// TIA Portal V20 export
// export: Created 2025-12-01T14:57:12.8919751Z, ExportSetting None, DisplayName Totally Integrated Automation Portal, DisplayVersion V20 Update 3, DisplayName TIA Portal Openness, DisplayVersion V20 Update 3, DisplayName TIA Portal Version Control Interface, DisplayVersion V20 Update 3, DisplayName STEP 7 Professional, DisplayVersion V20 Update 3, DisplayName STEP 7 Safety, DisplayVersion V20 Update 2, DisplayName WinCC Basic/Comfort/Advanced, DisplayVersion V20 Update 3, DisplayName WinCC Professional, DisplayVersion V20 Update 3, DisplayName WinCC Unified, DisplayVersion V20 Update 3
FUNCTION "FC811_EventosGenerados" : Void   // FC811, LAD
TITLE = "EventosGenerados" - Se generar la lista de Eventos a Emitir
{ S7_Optimized_Access := 'FALSE' }
AUTHOR : TRACKING
NAME : 20160407
VERSION : 4.2
// - Inicializaciones
// - Mirar si se pueden generar eventos
// - Generar eventos de las UT's
// - Generar eventos de los dispositivos
// - Generar eventos de las Mesas
// stored: AutoNumber false, SetENOAutomatically false
   VAR_INPUT
      NumJdT : UInt;
   END_VAR
   VAR_TEMP
      DBEventos : Word;   // Num. DB de eventos generados
      NumDBEventos : UInt;
      P_Eventos : DWord;   // Puntero al DB de Eventos Generados
      MaxBytes : UInt;
      InicioBucleMesas : UInt;
      FinalBucleMesas : UInt;
      NumBytes : UInt;   // Numero de Bytes a Emitir
      P_Temporal : DWord;
      NumMesa : UInt;   // Numero de Mesa a mirar
      IndiceEtiqueta : UInt;
      NumeroUT : UInt;   // Numero de UT a mirar
      EventoUT : UInt;   // Numero de Evento Generado en la UT
      EventoDispositivo : UInt;   // Numero de Evento Genarado en el Dispositivo
      NivelPantalla : UInt;   // Numero de nivel de pantalla
      Convertir : UInt;
      Conversion : DWord;
      Valor : UDInt;
      Offset : UInt;
      Proceso : UInt;
      ResultadoProceso : UInt;
      ValorReturn : Int;
      MesaDeJDT02 : Bool;
      JDT02_Activo : Bool;
      DispoDeJDT02 : Bool;
   END_VAR
BEGIN

NETWORK
TITLE = Inicializaciones
// - Inicializar las variables de los DB's
////////////////////////////////////////////////////////////////////////////////
////////////////////////////////////////////////////////////////////////////////
/// Inicio Que conexion es de JDT

      SET;
      R     #JDT02_Activo;
      L     "JDT1_NDB_EventosEmi";
      T     #DBEventos;
      T     #NumDBEventos;
      L     "JDT2_MaxBytes";
      T     #MaxBytes;

      L     "JDT1_InicioBucleMesas";  // Tamaño Bucles
      T     #InicioBucleMesas;
      L     "JDT1_FinalBucleMesas";
      T     #FinalBucleMesas;

      L     #NumJdT;
      L     2;
      <>I;
      JC    NoJDT02;

      SET;
      S     #JDT02_Activo;
      L     "JDT2_NDB_EventosEmi";
      T     #DBEventos;
      T     #NumDBEventos;
      L     "JDT2_MaxBytes";
      T     #MaxBytes;

      L     "JDT2_InicioBucleMesas";  // Tamaño Bucles
      T     #InicioBucleMesas;
      L     "JDT2_FinalBucleMesas";
      T     #FinalBucleMesas;

NoJDT02:NOP   0;

/// FIn Que conexion es de JDT
////////////////////////////////////////////////////////////////////////////////
////////////////////////////////////////////////////////////////////////////////



NETWORK
TITLE = Mirar si se pueden generar eventos
// - Inicializo el Numero de Bytes y el puntero del DB de Eventos Generados
// - Calcula el Tamaño de bytes que hay en el DB de Eventos Genardos
// - Comprobamos si hay sitio para Eventos
////////////////////////////////////////////////////////////////////////////////
// Inicializo el Numero de Bytes y el puntero del DB Eventos Generados

      L     0;
      T     #NumBytes;  // Inicializo el numero de Bytes
      LAR2;  // Inicializo el puntero de Eventos Generados

////////////////////////////////////////////////////////////////////////////////
// Calcula el tamaño de bytes que hay en el DB Eventos Generados

      OPN   DB [#DBEventos];

InicioBucleBusquedaFin_BufferEventos:NOP   0;
      L     DBB [AR2, P#0.0];
      L     0;
      ==I;
      JC    FinBucleBusquedaFin_BufferEventos;  // Buscamos el final del DB = 0

      +AR2  P#1.0;
      JU    InicioBucleBusquedaFin_BufferEventos;

FinBucleBusquedaFin_BufferEventos:NOP   0;
      TAR2;  // Guardo el puntero
      T     #P_Eventos;  // Sacamos el NumBytes Escritos
      SRD   3;
      T     #NumBytes;

////////////////////////////////////////////////////////////////////////////////
// Comprobamos si hay sitio para mas Eventos

      L     #NumBytes;  // Miramos si hay sitio
      L     #MaxBytes;  // Max. que se pueden emitir, parametro
      >I;
      JC    FinalFuncion;  // No se pueden generar más eventos



NETWORK
TITLE = Generar Eventos de las UT's
// - Recorrer todas las Mesas Buscando UT'que necesiten generar Eventos
//   Dos bucles anidados Mesas y UT's dentro de las Mesas ( No se hace)
// - Recorrer todas las UT's (Se hace
////////////////////////////////////////////////////////////////////////////////
////////////////////////////////////////////////////////////////////////////////
////////////////////////////////////////////////////////////////////////////////
// Recorrer todas las Mesas

      L     #InicioBucleMesas;
      T     #NumMesa;

InicioBucleMesa_EventosUT:NOP   0;
////////////////////////////////////////////////////////////////////////////////
/// Mirar Si pertenece al JDT

      SET;
      X     "DB850_DefinicionMesas".Mesa[#NumMesa].ConfigMesa.MesaDeJDT02;
      XN    #JDT02_Activo;  // JDT01 o JDT02 ?
      =     #MesaDeJDT02;

      SET;
      AN    #MesaDeJDT02;
      JC    ContinuarBucleMesa_EventosUT;

////////////////////////////////////////////////////////////////////////////////
// Mirar si esta definido como mesa de tracking

      SET;
      AN    "DB850_DefinicionMesas".Mesa[#NumMesa].ConfigMesa.MesaPaso;
      AN    "DB850_DefinicionMesas".Mesa[#NumMesa].ConfigMesa.MesaCruce;
      AN    "DB850_DefinicionMesas".Mesa[#NumMesa].ConfigMesa.MesaMultiplesDestinos;
      JC    ContinuarBucleMesa_EventosUT;


////////////////////////////////////////////////////////////////////////////////

      L     "DB810_ColasMesas".Colas[#NumMesa].UT_PrimeraMesa;
      T     #NumeroUT;

      L     #NumeroUT;
      L     0;
      ==I;
      JC    ContinuarBucleMesa_EventosUT;  // No hay UT's en la Mesa


////////////////////////////////////////////////////////////////////////////////
// --- Recorrer todas las UT's de la Mesa
InicioBucleUT_EventosUT:NOP   0;

      L     "DB812_UTs_Control".UT[#NumeroUT].EstadoEventoAGenerar;
      T     #EventoUT;  // Para ver si hay Evento de UT

      L     #EventoUT;  // Mirar si hay evento a generar
      L     100;
      >=I;
      JC    Generar_EventosUT;  // Si es >= 100 Hay evento a generar


////////////////////////////////////////////////////////////////////////////////
ContinuarBucleUT_EventosUT:NOP   0;
      L     "DB812_UTs_Control".UT[#NumeroUT].UT_SiguienteMesa;
      T     #NumeroUT;

      L     #NumeroUT;
      L     0;
      ==I;
      JC    ContinuarBucleMesa_EventosUT;  // No hay mas UT's en la Mesa

      JU    InicioBucleUT_EventosUT;  // Seguir recorriendo la Mesa


////////////////////////////////////////////////////////////////////////////////
// --- Continuar recorriendo el resto de Mesas
ContinuarBucleMesa_EventosUT:NOP   0;
      L     #NumMesa;
      L     #FinalBucleMesas;
      >=I;
      JC    EventosMesa;  // Ya no hay más UT's, recorrer dispositivos

      L     #NumMesa;  // +1, Para la Siguiente UT
      L     1;
      +I;
      T     #NumMesa;

      JU    InicioBucleMesa_EventosUT;  // Ir a mirar la siguiente UT


////////////////////////////////////////////////////////////////////////////////
// Comprobacion del tamaño del DB de Eventos Generados
FinBucles_EventosUT:NOP   0;
      TAR2;
      T     #P_Eventos;
      SRD   3;
      T     #NumBytes;

      L     #NumBytes;  // Miramos si hay sitio
      L     #MaxBytes;
      >I;
      JC    FinalFuncion;  // No se pueden generar más eventos
      JU    ContinuarBucleUT_EventosUT;  // Seguir con las UT's



NETWORK
TITLE = Formatear Eventos de las UTs - Distribucion
Generar_EventosUT:NOP   0;

////////////////////////////////////////////////////////////////////////////////
////////////////////////////////////////////////////////////////////////////////
// -- Formateo del Evento LOCA - Diferentes Motivos (Normal, Reset, Galibo ...)
// -- Formateo del Evento RUT? - Diferentes (Reset, PLC, ...)
// -- Formateo del Evento RET! - Ausencia de la Mesa
// -- Formateo del Evento BOR! - Borrada UT del Sistema
// -- Formateo del Evento DATO - Refresco de Datos de la UT
// -- Formateo del Evento NUUT - Nueva UT en la Mesa
// -- Formateo del Evento DAT? - Peticion de Datos para la UT
// -- Formateo del Evento PEMB (Peticion de Datos de Embandejado de la UT)
////////////////////////////////////////////////////////////////////////////////
////////////////////////////////////////////////////////////////////////////////
// Distribucion para Eventos de las UT's

      L     #EventoUT;  // Formateo del evento
      L     100;  // Presencia Normal
      ==I;
      JC    GenerarEvento_LOCA_EventosUT;

      L     #EventoUT;  // Formateo del evento
      L     101;  // Presencia de Reset
      ==I;
      JC    GenerarEvento_LOCA_EventosUT;

      L     #EventoUT;  // Formateo del evento
      L     102;  // Presencia de Galibo
      ==I;
      JC    GenerarEvento_LOCA_EventosUT;

      L     #EventoUT;  // Formateo del evento
      L     103;  // Ausencia
      ==I;
      JC    GenerarEvento_RET_EventosUT;

      L     #EventoUT;  // Formateo del evento
      L     110;  // Refresco de datos de la UT
      ==I;
      JC    GenerarEvento_DATO_EventoUT;

      L     #EventoUT;  // Formateo del evento
      L     121;  // Peticion de Ruta por MOTIVO --> Reset
      ==I;
      JC    GenerarEvento_RUT_EventoUT;

      L     #EventoUT;  // Formateo del evento
      L     122;  // Peticion de Ruta por MOTIVO --> Bloqueo
      ==I;
      JC    GenerarEvento_RUT_EventoUT;

      L     #EventoUT;  // Formateo del evento
      L     123;  // Peticion de Ruta por MOTIVO --> Llegada a su Destino
      ==I;
      JC    GenerarEvento_RUT_EventoUT;

      L     #EventoUT;  // Formateo del evento
      L     124;  // Peticion de Ruta por MOTIVO --> No tiene Destino
      ==I;
      JC    GenerarEvento_RUT_EventoUT;

      L     #EventoUT;  // Formateo del evento
      L     125;  // Peticion de Ruta por MOTIVO --> Fuera de Ruta
      ==I;
      JC    GenerarEvento_RUT_EventoUT;

      L     #EventoUT;  // Formateo del evento
      L     126;  // Peticion de Ruta por MOTIVO --> Robo de Garra a Elevador
      ==I;
      JC    GenerarEvento_RUT_EventoUT;

      L     #EventoUT;  // Formateo del evento
      L     131;  // Borrar la UT de la Base de datos
      ==I;
      JC    GenerarEvento_BOR_EventosUT;

      L     #EventoUT;  // Formateo del evento
      L     132;  // Nueva UT en la BD
      ==I;
      JC    GenerarEvento_NUUT_EventosUT;

      L     #EventoUT;  // Formateo del evento
      L     141;  // Peticion de datos para la UT
      ==I;
      JC    GenerarEvento_DAT_EventosUT;

      L     #EventoUT;  // Formateo del evento
      L     145;  // Chequeo de la UT >>> Por Reset
      ==I;
      JC    GenerarEvento_CHE_EventosUT;

      L     #EventoUT;  // Formateo del evento     // Fecha 2019 01 18
      L     161;  // Peticion de datos de Embandejado para la UT
      ==I;
      JC    GenerarEvento_PEMB_EventosUT;


////////////////////////////////////////////////////////////////////////////////
////////////////////////////////////////////////////////////////////////////////
////////////////////////////////////////////////////////////////////////////////
// --- Dar por formateado el Evento

      L     0;  // 0 - Dar por Tratado
      T     "DB812_UTs_Control".UT[#NumeroUT].EstadoEventoAGenerar;

      JU    FinBucles_EventosUT;

// Fin de la distribucion para generar los eventos
////////////////////////////////////////////////////////////////////////////////
////////////////////////////////////////////////////////////////////////////////
////////////////////////////////////////////////////////////////////////////////



NETWORK
TITLE = ---- Eventos de UT - Esta en Mesa - LOCA
// - Distribucion para Eventos de las UT's
// - Formateo de Eventos
//   - Evento LOCA (Cambio de Mesa de la UT
//   - Evento RUT? (Petición de Ruta para la UT)
//   - Evento NUUT (Nueva UT en la instalacion)
//   - Evento DATO (Cambio de de datos de la UT)
//   - Evento BOR! (UT Borrada de la Base de datos)
//   - Evento DAT? (Peticion de datos de la UT)
//   - Evento RET! (Retirada de la UT)
GenerarEvento_LOCA_EventosUT:NOP   0;

////////////////////////////////////////////////////////////////////////////////
////////////////////////////////////////////////////////////////////////////////
////////////////////////////////////////////////////////////////////////////////
// -- Formateo del Evento LOCA - Diferentes Motivos (Normal, Reset, Galibo ...)

      L     #P_Eventos;
      LAR2;  // Puntero al DB de Eventos Generados

      TAR2;  // Mirar si es el primer evento de la lista
      L     0;
      ==I;
      JC    InicioBuffer_LOCA_EventosUT;  // Es el primero

      OPN   DB [#DBEventos];  // Hay que añadir si no es el primer evento
      L     ',';  // Separador entre eventos ','
      T     DBB [AR2, P#0.0];
      +AR2  P#1.0;

InicioBuffer_LOCA_EventosUT:NOP   0;
      OPN   DB [#DBEventos];  // DB de Eventos Generados (A Emitir)
      L     '{';  // Inicio de Evento '{'
      T     DBB [AR2, P#0.0];
      +AR2  P#1.0;


////////////////////////////////////////////////////////////////////////////////
      L     'LOCA';  // Evento 'LOCA'
      T     DBD [AR2, P#0.0];
      +AR2  P#4.0;

      L     '[';  // Evento - Atributo Mckey '[MCKY]'
      T     DBB [AR2, P#0.0];
      L     'MCKY';
      T     DBD [AR2, P#1.0];
      L     ']';  // Evento - Atributo Mckey '[MCKY]'
      T     DBB [AR2, P#5.0];
      +AR2  P#6.0;

      L     "DB812_UTs_Control".UT[#NumeroUT].Mckey;
      T     #Valor;

// --- Convertir Valor a ASCII - Mckey
      TAR2;
      SRD   3;
      T     #NumBytes;  // Miro que offset tiene la String

      CALL  "FC893_Obtener_StringDelAtributo"
      ( DB_String := #NumDBEventos,
        OffsetIni := #NumBytes,
        Valor     := #Valor,
        OffsetFin := #Offset
      );  // Llamo a ObtenerStrinAtributo

      L     #Offset;
      SLD   3;
      LAR2;  // Recupero que offset tiene la String

// --- Ya esta convertido el Valor a ASCI - Fin Mckey


////////////////////////////////////////////////////////////////////////////////
      OPN   DB [#DBEventos];
      L     '[';  // Evento - Atributo Mesa Actual '[MESA]'
      T     DBB [AR2, P#0.0];
      L     'MESA';
      T     DBD [AR2, P#1.0];
      L     ']';
      T     DBB [AR2, P#5.0];
      +AR2  P#6.0;

      L     "DB812_UTs_Control".UT[#NumeroUT].MesaActual;
      T     #Valor;

// --- Convertir Valor a ASCII -  Mesa Actual
      TAR2;
      SRD   3;
      T     #NumBytes;  // Miro que offset tiene la String

      CALL  "FC893_Obtener_StringDelAtributo"
      ( DB_String := #NumDBEventos,
        OffsetIni := #NumBytes,
        Valor     := #Valor,
        OffsetFin := #Offset
      );  // Llamo a ObtenerStrinAtributo

      L     #Offset;
      SLD   3;
      LAR2;  // Recupero que offset tiene la String

// --- Ya esta convertido el Valor a ASCI - Fin Mesa Actual


////////////////////////////////////////////////////////////////////////////////
// --- Final del Formateo del Evento ---

      OPN   DB [#DBEventos];  // DB de Eventos Generados (A Emitir)
      L     '}';  // Fin de Evento '}'
      T     DBB [AR2, P#0.0];
      +AR2  P#1.0;



////////////////////////////////////////////////////////////////////////////////
////////////////////////////////////////////////////////////////////////////////
////////////////////////////////////////////////////////////////////////////////
// --- Dar por formateado el Evento

      L     0;  // 0 - Dar por Tratado
      T     "DB812_UTs_Control".UT[#NumeroUT].EstadoEventoAGenerar;

////////////////////////////////////////////////////////////////////////////////
/// Hay que Pedir Datos
      SET;
      AN    "DB812_UTs_Control".UT[#NumeroUT].AtributosDeLaUT.PeticionDeDatos;
      JC    NoPedirDatos_LOCA_EventosUT;

      L     141;
      T     "DB812_UTs_Control".UT[#NumeroUT].EstadoEventoAGenerar;

NoPedirDatos_LOCA_EventosUT:NOP   0;

////////////////////////////////////////////////////////////////////////////////
/// Hay que Generar mas Eventos
      L     #EventoUT;  // Formateo del evento
      L     100;  // Presencia Normal
      ==I;
      JC    FinBucles_EventosUT;

////////////////////////////////////////////////////////////////////////////////
/// Es de Reset de Pantalla, Auto Generar Nuevo Evento
      L     121;  // 121 - Generar evento de Pedir Ruta (Por Reset)
      T     "DB812_UTs_Control".UT[#NumeroUT].EstadoEventoAGenerar;

      L     #EventoUT;  // Formateo del evento
      L     101;  // Presencia de Reset
      ==I;
      JC    FinBucles_EventosUT;


////////////////////////////////////////////////////////////////////////////////
/// Es de Galibo, Auto Generar Nuevo Evento
      L     110;  // Enviar datos de UT
      T     "DB812_UTs_Control".UT[#NumeroUT].EstadoEventoAGenerar;

      JU    FinBucles_EventosUT;

// Fin del Evento LOCA
////////////////////////////////////////////////////////////////////////////////
////////////////////////////////////////////////////////////////////////////////
////////////////////////////////////////////////////////////////////////////////



NETWORK
TITLE = ---- Evento de UT - Peticion de Ruta - RUT?
GenerarEvento_RUT_EventoUT:NOP   0;

////////////////////////////////////////////////////////////////////////////////
////////////////////////////////////////////////////////////////////////////////
////////////////////////////////////////////////////////////////////////////////
////////////////////////////////////////////////////////////////////////////////
// -- Formateo del Evento RUT? - Diferentes (Reset, PLC, ...)

      L     #P_Eventos;
      LAR2;  // Puntero al DB de Eventos Generados

      TAR2;  // Mirar si es el primer evento de la lista
      L     0;
      ==I;
      JC    InicioBuffer_RUT_EventosUT;  // Es el primero

      OPN   DB [#DBEventos];  // Hay que añadir si no es el primer evento
      L     ',';  // Separador entre eventos ','
      T     DBB [AR2, P#0.0];
      +AR2  P#1.0;

InicioBuffer_RUT_EventosUT:NOP   0;
      OPN   DB [#DBEventos];  // DB de Eventos Generados (A Emitir)
      L     '{';  // Inicio de Evento '{'
      T     DBB [AR2, P#0.0];
      +AR2  P#1.0;

      L     'RUT?';  // Evento 'RUT?'
      T     DBD [AR2, P#0.0];
      +AR2  P#4.0;


////////////////////////////////////////////////////////////////////////////////
      L     '[';  // Evento - Atributo Mckey '[MCKEY]'
      T     DBB [AR2, P#0.0];
      L     'MCKY';
      T     DBD [AR2, P#1.0];
      L     ']';
      T     DBB [AR2, P#5.0];
      +AR2  P#6.0;

      L     "DB812_UTs_Control".UT[#NumeroUT].Mckey;
      T     #Valor;

// --- Convertir Valor a ASCII - Mckey
      TAR2;
      SRD   3;
      T     #NumBytes;  // Miro que offset tiene la String

      CALL  "FC893_Obtener_StringDelAtributo"
      ( DB_String := #NumDBEventos,
        OffsetIni := #NumBytes,
        Valor     := #Valor,
        OffsetFin := #Offset
      );  // Llamo a ObtenerStrinAtributo

      L     #Offset;
      SLD   3;
      LAR2;  // Recupero que offset tiene la String

// --- Ya esta convertido el Valor a ASCI - Fin Mckey


////////////////////////////////////////////////////////////////////////////////
      OPN   DB [#DBEventos];
      L     '[';  // Evento - Atributo Mesa Actual '[MESA]'
      T     DBB [AR2, P#0.0];
      L     'MESA';
      T     DBD [AR2, P#1.0];
      L     ']';
      T     DBB [AR2, P#5.0];
      +AR2  P#6.0;

      L     "DB812_UTs_Control".UT[#NumeroUT].MesaActual;
      T     #Valor;

// --- Convertir Valor a ASCII -  Mesa Actual
      TAR2;
      SRD   3;
      T     #NumBytes;  // Miro que offset tiene la String

      CALL  "FC893_Obtener_StringDelAtributo"
      ( DB_String := #NumDBEventos,
        OffsetIni := #NumBytes,
        Valor     := #Valor,
        OffsetFin := #Offset
      );  // Llamo a ObtenerStrinAtributo

      L     #Offset;
      SLD   3;
      LAR2;  // Recupero que offset tiene la String

// --- Ya esta convertido el Valor a ASCI - Fin Mesa Actual


////////////////////////////////////////////////////////////////////////////////
      OPN   DB [#DBEventos];
      L     '[';  // Evento - Atributo Motivo '[MOTI]'
      T     DBB [AR2, P#0.0];
      L     'MOTI';
      T     DBD [AR2, P#1.0];
      L     ']';
      T     DBB [AR2, P#5.0];
      +AR2  P#6.0;

      L     #EventoUT;  // Poner Motivo
      T     #Convertir;
      CALL  "FC895_Obtener_EtiquetaDeValor"
      ( ValorEvento    := #Convertir,
        EtiquetaEvento := #Conversion
      );

      OPN   DB [#DBEventos];
      L     #Conversion;
      T     DBD [AR2, P#0.0];
      +AR2  P#4.0;


////////////////////////////////////////////////////////////////////////////////
// --- Final del Formateo del Evento ---

      OPN   DB [#DBEventos];  // DB de Eventos Generados (A Emitir)
      L     '}';  // Fin de Evento '}'
      T     DBB [AR2, P#0.0];
      +AR2  P#1.0;


////////////////////////////////////////////////////////////////////////////////
////////////////////////////////////////////////////////////////////////////////
////////////////////////////////////////////////////////////////////////////////
// Dar por formateado el Evento

      L     0;  // 0 - Dar por Tratado
      T     "DB812_UTs_Control".UT[#NumeroUT].EstadoEventoAGenerar;

////////////////////////////////////////////////////////////////////////////////
/// Hay que Pedir Datos
      SET;
      AN    "DB812_UTs_Control".UT[#NumeroUT].AtributosDeLaUT.PeticionDeDatos;
      JC    NoPedirDatos_RUT_EventosUT;

      L     141;
      T     "DB812_UTs_Control".UT[#NumeroUT].EstadoEventoAGenerar;

NoPedirDatos_RUT_EventosUT:NOP   0;


////////////////////////////////////////////////////////////////////////////////
      JU    FinBucles_EventosUT;


// Fin del Evento RUT?
////////////////////////////////////////////////////////////////////////////////
////////////////////////////////////////////////////////////////////////////////
////////////////////////////////////////////////////////////////////////////////



NETWORK
TITLE = ---- Eventos de UT - Ausencia de la Mesa - RET!
GenerarEvento_RET_EventosUT:NOP   0;

////////////////////////////////////////////////////////////////////////////////
////////////////////////////////////////////////////////////////////////////////
////////////////////////////////////////////////////////////////////////////////
////////////////////////////////////////////////////////////////////////////////
// -- Formateo del Evento RET! - Ausencia de la Mesa

      L     #P_Eventos;
      LAR2;  // Puntero al DB de Eventos Generados

      TAR2;  // Mirar si es el primer evento de la lista
      L     0;
      ==I;
      JC    InicioBuffer_RET_EventosUT;  // Es el primero

      OPN   DB [#DBEventos];  // Hay que añadir si no es el primer evento
      L     ',';  // Separador entre eventos ','
      T     DBB [AR2, P#0.0];
      +AR2  P#1.0;

InicioBuffer_RET_EventosUT:NOP   0;
      OPN   DB [#DBEventos];  // DB de Eventos Generados (A Emitir)
      L     '{';  // Inicio de Evento '{'
      T     DBB [AR2, P#0.0];
      +AR2  P#1.0;

      L     'RET!';  // Evento 'RET!'
      T     DBD [AR2, P#0.0];
      +AR2  P#4.0;


////////////////////////////////////////////////////////////////////////////////
      L     '[';  // Evento - Atributo Mckey '[MCKY]'
      T     DBB [AR2, P#0.0];
      L     'MCKY';
      T     DBD [AR2, P#1.0];
      L     ']';
      T     DBB [AR2, P#5.0];
      +AR2  P#6.0;

      L     "DB812_UTs_Control".UT[#NumeroUT].Mckey;
      T     #Valor;

// --- Convertir Valor a ASCII - Mckey
      TAR2;
      SRD   3;
      T     #NumBytes;  // Miro que offset tiene la String

      CALL  "FC893_Obtener_StringDelAtributo"
      ( DB_String := #NumDBEventos,
        OffsetIni := #NumBytes,
        Valor     := #Valor,
        OffsetFin := #Offset
      );  // Llamo a ObtenerStrinAtributo

      L     #Offset;
      SLD   3;
      LAR2;  // Recupero que offset tiene la String

// --- Ya esta convertido el Valor a ASCI - Fin Mckey


////////////////////////////////////////////////////////////////////////////////
      OPN   DB [#DBEventos];
      L     '[';  // Evento - Atributo Mesa Actual '[MESA]'
      T     DBB [AR2, P#0.0];
      L     'MESA';
      T     DBD [AR2, P#1.0];
      L     ']';
      T     DBB [AR2, P#5.0];
      +AR2  P#6.0;

      L     "DB812_UTs_Control".UT[#NumeroUT].MesaActual;
      T     #Valor;

// --- Convertir Valor a ASCII -  Mesa Actual
      TAR2;
      SRD   3;
      T     #NumBytes;  // Miro que offset tiene la String

      CALL  "FC893_Obtener_StringDelAtributo"
      ( DB_String := #NumDBEventos,
        OffsetIni := #NumBytes,
        Valor     := #Valor,
        OffsetFin := #Offset
      );  // Llamo a ObtenerStrinAtributo

      L     #Offset;
      SLD   3;
      LAR2;  // Recupero que offset tiene la String

// --- Ya esta convertido el Valor a ASCI - Fin Mesa Actual


////////////////////////////////////////////////////////////////////////////////
// --- Final del Formato del Evento ---

      OPN   DB [#DBEventos];  // DB de Eventos Generados (A Emitir)
      L     '}';  // Fin de Evento '}'
      T     DBB [AR2, P#0.0];
      +AR2  P#1.0;


////////////////////////////////////////////////////////////////////////////////
////////////////////////////////////////////////////////////////////////////////
////////////////////////////////////////////////////////////////////////////////
////////////////////////////////////////////////////////////////////////////////
// Dar por formateado el Evento

      L     0;  // 0 - Dar por Tratado
      T     "DB812_UTs_Control".UT[#NumeroUT].EstadoEventoAGenerar;

      JU    FinBucles_EventosUT;

// Fin del formateo del Evento RET!
////////////////////////////////////////////////////////////////////////////////
////////////////////////////////////////////////////////////////////////////////
////////////////////////////////////////////////////////////////////////////////
////////////////////////////////////////////////////////////////////////////////



NETWORK
TITLE = ---- Evento de UT - Borrar la UT de la Mesa - BOR!
GenerarEvento_BOR_EventosUT:NOP   0;

////////////////////////////////////////////////////////////////////////////////
////////////////////////////////////////////////////////////////////////////////
////////////////////////////////////////////////////////////////////////////////
////////////////////////////////////////////////////////////////////////////////
// -- Formateo del Evento BOR! - Borrada UT del Sistema


      L     #P_Eventos;
      LAR2;  // Puntero al DB de Eventos Generados

      TAR2;  // Mirar si es el primer evento de la lista
      L     0;
      ==I;
      JC    InicioBuffer_BOR_EventosUT;  // Es el primero

      OPN   DB [#DBEventos];  // Hay que añadir si no es el primer evento
      L     ',';  // Separador entre eventos ','
      T     DBB [AR2, P#0.0];
      +AR2  P#1.0;

InicioBuffer_BOR_EventosUT:NOP   0;
      OPN   DB [#DBEventos];  // DB de Eventos Generados (A Emitir)
      L     '{';  // Inicio de Evento '{'
      T     DBB [AR2, P#0.0];
      +AR2  P#1.0;

      L     'BOR!';  // Evento 'BOR!'
      T     DBD [AR2, P#0.0];
      +AR2  P#4.0;


////////////////////////////////////////////////////////////////////////////////
      L     '[';  // Evento - Atributo Mckey '[MCKY]'
      T     DBB [AR2, P#0.0];
      L     'MCKY';
      T     DBD [AR2, P#1.0];
      L     ']';
      T     DBB [AR2, P#5.0];
      +AR2  P#6.0;

      L     "DB812_UTs_Control".UT[#NumeroUT].Mckey;
      T     #Valor;

// --- Convertir Valor a ASCII - Mckey
      TAR2;
      SRD   3;
      T     #NumBytes;  // Miro que offset tiene la String

      CALL  "FC893_Obtener_StringDelAtributo"
      ( DB_String := #NumDBEventos,
        OffsetIni := #NumBytes,
        Valor     := #Valor,
        OffsetFin := #Offset
      );  // Llamo a ObtenerStrinAtributo

      L     #Offset;
      SLD   3;
      LAR2;  // Recupero que offset tiene la String

// --- Ya esta convertido el Valor a ASCI - Fin Mckey


////////////////////////////////////////////////////////////////////////////////
      OPN   DB [#DBEventos];
      L     '[';  // Evento - Atributo Mesa Actual 'MESA'
      T     DBB [AR2, P#0.0];
      L     'MESA';
      T     DBD [AR2, P#1.0];
      L     ']';
      T     DBB [AR2, P#5.0];
      +AR2  P#6.0;

      L     "DB812_UTs_Control".UT[#NumeroUT].MesaActual;
      T     #Valor;

// --- Convertir Valor a ASCII -  Mesa Actual
      TAR2;
      SRD   3;
      T     #NumBytes;  // Miro que offset tiene la String

      CALL  "FC893_Obtener_StringDelAtributo"
      ( DB_String := #NumDBEventos,
        OffsetIni := #NumBytes,
        Valor     := #Valor,
        OffsetFin := #Offset
      );  // Llamo a ObtenerStrinAtributo

      L     #Offset;
      SLD   3;
      LAR2;  // Recupero que offset tiene la String

// --- Ya esta convertido el Valor a ASCI - Fin Mesa Actual


////////////////////////////////////////////////////////////////////////////////
// --- Final del Formato del Evento ---

      OPN   DB [#DBEventos];  // DB de Eventos Generados (A Emitir)
      L     '}';  // Fin de Evento '}'
      T     DBB [AR2, P#0.0];
      +AR2  P#1.0;


////////////////////////////////////////////////////////////////////////////////
////////////////////////////////////////////////////////////////////////////////
////////////////////////////////////////////////////////////////////////////////
////////////////////////////////////////////////////////////////////////////////
// Borrar la UT de la Base de datos

      CALL  "FC722_EliminarUT_DeMesa"
      ( NumeroUT := #NumeroUT
      );

      JU    FinBucles_EventosUT;

// Fin del formateo del Evento BOR!
////////////////////////////////////////////////////////////////////////////////
////////////////////////////////////////////////////////////////////////////////
////////////////////////////////////////////////////////////////////////////////
////////////////////////////////////////////////////////////////////////////////



NETWORK
TITLE = ---- Evento de UT - Nueva UT en la Mesa - NUUT
GenerarEvento_NUUT_EventosUT:NOP   0;

////////////////////////////////////////////////////////////////////////////////
////////////////////////////////////////////////////////////////////////////////
////////////////////////////////////////////////////////////////////////////////
////////////////////////////////////////////////////////////////////////////////
// -- Formateo del Evento NUUT - Nueva UT en la Mesa

      L     #P_Eventos;
      LAR2;  // Puntero al DB de Eventos Generados

      TAR2;  // Mirar si es el primer evento de la lista
      L     0;
      ==I;
      JC    InicioBuffer_NUUT_EventosUT;  // Es el primero

      OPN   DB [#DBEventos];  // Hay que añadir si no es el primer evento
      L     ',';  // Separador entre eventos ','
      T     DBB [AR2, P#0.0];
      +AR2  P#1.0;

InicioBuffer_NUUT_EventosUT:NOP   0;
      OPN   DB [#DBEventos];  // DB de Eventos Generados (A Emitir)
      L     '{';  // Inicio de Evento '{'
      T     DBB [AR2, P#0.0];
      +AR2  P#1.0;

      L     'NUUT';  // Evento  'NUUT'
      T     DBD [AR2, P#0.0];
      +AR2  P#4.0;


////////////////////////////////////////////////////////////////////////////////
      OPN   DB [#DBEventos];
      L     '[';  // Evento - Atributo Mesa Actual '[MESA]'
      T     DBB [AR2, P#0.0];
      L     'MESA';
      T     DBD [AR2, P#1.0];
      L     ']';
      T     DBB [AR2, P#5.0];
      +AR2  P#6.0;

      L     "DB812_UTs_Control".UT[#NumeroUT].MesaActual;
      T     #Valor;

// --- Convertir Valor a ASCII -  Mesa Actual
      TAR2;
      SRD   3;
      T     #NumBytes;  // Miro que offset tiene la String

      CALL  "FC893_Obtener_StringDelAtributo"
      ( DB_String := #NumDBEventos,
        OffsetIni := #NumBytes,
        Valor     := #Valor,
        OffsetFin := #Offset
      );  // Llamo a ObtenerStrinAtributo

      L     #Offset;
      SLD   3;
      LAR2;  // Recupero que offset tiene la String

// --- Ya esta convertido el Valor a ASCI - Fin Mesa Actual


////////////////////////////////////////////////////////////////////////////////
////////////////////////////////////////////////////////////////////////////////
////////////////////////////////////////////////////////////////////////////////
////////////////////////////////////////////////////////////////////////////////
// --- Caracteristicas de la UT a Emitir


////////////////////////////////////////////////////////////////////////////////
// --- Atributo de ALTURA COTA (Si es necesario) ---
      SET;
      AN    "DB850_DefinicionMesas".Mesa[#NumMesa].AtributosGalibo_DeEvento.Cota_Altura;  // Tiene Cota Altura ?
      JC    CotaAltura_NUNUT_EventosUT;

      L     "DB815_UTs_Datos".UT[#NumeroUT].CotaAltura;
      T     #Valor;

      OPN   DB [#DBEventos];
      L     '[';  // Evento - Atributo Altura Cota '[ALTO]'
      T     DBB [AR2, P#0.0];
      L     'COTA';
      T     DBD [AR2, P#1.0];
      L     ']';
      T     DBB [AR2, P#5.0];
      +AR2  P#6.0;

// --- Convertir Valor a ASCII -  Altura Cota
      TAR2;
      SRD   3;
      T     #NumBytes;  // Miro que offset tiene la String

      CALL  "FC893_Obtener_StringDelAtributo"
      ( DB_String := #NumDBEventos,
        OffsetIni := #NumBytes,
        Valor     := #Valor,
        OffsetFin := #Offset
      );  // Llamo a ObtenerStrinAtributo

      L     #Offset;
      SLD   3;
      LAR2;  // Recupero que offset tiene la String

// --- Ya esta convertido el Valor a ASCI - Fin Altura Cota
CotaAltura_NUNUT_EventosUT:NOP   0;


////////////////////////////////////////////////////////////////////////////////
////////////////////////////////////////////////////////////////////////////////
////////////////////////////////////////////////////////////////////////////////
////////////////////////////////////////////////////////////////////////////////
// --- Atributo de GALIBO (ALTO, ANCH, LARG, REMO) (Si es necesario) ---
      SET;
      AN    "DB850_DefinicionMesas".Mesa[#NumMesa].AtributosGalibo_DeEvento.Altura;  // Tiene Altura ?
      JC    CodigoAltura_NUUT_EventosUT;

      OPN   DB [#DBEventos];
      L     '[';  // Evento - Atributo Galibo Altura '[ALTO]'
      T     DBB [AR2, P#0.0];
      L     'ALTO';
      T     DBD [AR2, P#1.0];
      L     ']';
      T     DBB [AR2, P#5.0];
      +AR2  P#6.0;

      L     "DB815_UTs_Datos".UT[#NumeroUT].GaliboAltura;
      T     #Valor;

// --- Convertir Valor a ASCII -  Alto
      TAR2;
      SRD   3;
      T     #NumBytes;  // Miro que offset tiene la String

      CALL  "FC893_Obtener_StringDelAtributo"
      ( DB_String := #NumDBEventos,
        OffsetIni := #NumBytes,
        Valor     := #Valor,
        OffsetFin := #Offset
      );  // Llamo a ObtenerStrinAtributo

      L     #Offset;
      SLD   3;
      LAR2;  // Recupero que offset tiene la String

// nieves inicio modificación emisión atributo VACI

//Comprobar si tenemos que emitir el evento

      SET;
      L     "DB815_UTs_Datos".UT[#NumeroUT].GaliboVacia;
      L     0;
      ==I;
      JC    CodigoAltura_NUUT_EventosUT;

      OPN   DB [#DBEventos];
      L     '[';  // Evento - Atributo Galibo Altura '[ALTO]'
      T     DBB [AR2, P#0.0];
      L     'VACI';
      T     DBD [AR2, P#1.0];
      L     ']';
      T     DBB [AR2, P#5.0];
      +AR2  P#6.0;

      L     "DB815_UTs_Datos".UT[#NumeroUT].GaliboVacia;
      L     1;
      -I;
      T     #Valor;

// --- Convertir Valor a ASCII -  VACIO
      TAR2;
      SRD   3;
      T     #NumBytes;  // Miro que offset tiene la String

      CALL  "FC893_Obtener_StringDelAtributo"
      ( DB_String := #NumDBEventos,
        OffsetIni := #NumBytes,
        Valor     := #Valor,
        OffsetFin := #Offset
      );  // Llamo a ObtenerStrinAtributo


      L     #Offset;
      SLD   3;
      LAR2;  // Recupero que offset tiene la String


// fin modificación atributo VACI

// --- Ya esta convertido el Valor a ASCI - Fin Alto
CodigoAltura_NUUT_EventosUT:NOP   0;


////////////////////////////////////////////////////////////////////////////////
      SET;
      AN    "DB850_DefinicionMesas".Mesa[#NumMesa].AtributosGalibo_DeEvento.Anchura;  // Tiene Anchura ?
      JC    CodigoAnchura_NUUT_EventosUT;

      OPN   DB [#DBEventos];
      L     '[';  // Evento - Atributo Galibo Anchura '[ANCH]'
      T     DBB [AR2, P#0.0];
      L     'ANCH';
      T     DBD [AR2, P#1.0];
      L     ']';
      T     DBB [AR2, P#5.0];
      +AR2  P#6.0;

      L     "DB815_UTs_Datos".UT[#NumeroUT].GaliboAnchura;
      T     #Valor;

// --- Convertir Valor a ASCII -  Anchura
      TAR2;
      SRD   3;
      T     #NumBytes;  // Miro que offset tiene la String

      CALL  "FC893_Obtener_StringDelAtributo"
      ( DB_String := #NumDBEventos,
        OffsetIni := #NumBytes,
        Valor     := #Valor,
        OffsetFin := #Offset
      );  // Llamo a ObtenerStrinAtributo

      L     #Offset;
      SLD   3;
      LAR2;  // Recupero que offset tiene la String

// --- Ya esta convertido el Valor a ASCI - Fin Anchura
CodigoAnchura_NUUT_EventosUT:NOP   0;


////////////////////////////////////////////////////////////////////////////////
      SET;
      AN    "DB850_DefinicionMesas".Mesa[#NumMesa].AtributosGalibo_DeEvento.Profundidad;  // Tiene Profundidad ?
      JC    CodigoLargura_NUUT_EventosUT;

      OPN   DB [#DBEventos];
      L     '[';  // Evento - Atributo Galibo Profuncidad '[PROF]'
      T     DBB [AR2, P#0.0];
      L     'PROF';
      T     DBD [AR2, P#1.0];
      L     ']';
      T     DBB [AR2, P#5.0];
      +AR2  P#6.0;

      L     "DB815_UTs_Datos".UT[#NumeroUT].GaliboProfundidad;
      T     #Valor;

// --- Convertir Valor a ASCII -  Profundidad
      TAR2;
      SRD   3;
      T     #NumBytes;  // Miro que offset tiene la String

      CALL  "FC893_Obtener_StringDelAtributo"
      ( DB_String := #NumDBEventos,
        OffsetIni := #NumBytes,
        Valor     := #Valor,
        OffsetFin := #Offset
      );  // Llamo a ObtenerStrinAtributo

      L     #Offset;
      SLD   3;
      LAR2;  // Recupero que offset tiene la String

// --- Ya esta convertido el Valor a ASCI - Fin Profundidad
CodigoLargura_NUUT_EventosUT:NOP   0;


////////////////////////////////////////////////////////////////////////////////
      SET;
      AN    "DB850_DefinicionMesas".Mesa[#NumMesa].AtributosGalibo_DeEvento.Remontado;  // Tiene Remontado ?
      JC    CodigoRemontado_NUUT_EventosUT;

      OPN   DB [#DBEventos];
      L     '[';  // Evento - Atributo Galibo Remontada '[REMO]'
      T     DBB [AR2, P#0.0];
      L     'REMO';
      T     DBD [AR2, P#1.0];
      L     ']';
      T     DBB [AR2, P#5.0];
      +AR2  P#6.0;

      L     "DB815_UTs_Datos".UT[#NumeroUT].GaliboRemontada;
      L     1;
      -I;
      L     W#16#30;
      +I;
      OPN   DB [#DBEventos];
      T     DBB [AR2, P#0.0];
      +AR2  P#1.0;

CodigoRemontado_NUUT_EventosUT:NOP   0;

////////////////////////////////////////////////////////////////////////////////
////////////////////////////////////////////////////////////////////////////////
////////////////////////////////////////////////////////////////////////////////
////////////////////////////////////////////////////////////////////////////////


////////////////////////////////////////////////////////////////////////////////
// --- Atributo de PESO (Si es necesario) ---
      SET;
      AN    "DB850_DefinicionMesas".Mesa[#NumMesa].AtributosGalibo_DeEvento.Peso;  // Tiene Peso ?
      JC    Peso_NUUT_EventoUT;

      L     "DB815_UTs_Datos".UT[#NumeroUT].Peso;
      T     #Valor;

      OPN   DB [#DBEventos];
      L     '[';  // Evento - Atributo Peso '[PESO]'
      T     DBB [AR2, P#0.0];
      L     'PESO';
      T     DBD [AR2, P#1.0];
      L     ']';
      T     DBB [AR2, P#5.0];
      +AR2  P#6.0;

// --- Convertir Valor a ASCII -  Peso
      TAR2;
      SRD   3;
      T     #NumBytes;  // Miro que offset tiene la String

      CALL  "FC893_Obtener_StringDelAtributo"
      ( DB_String := #NumDBEventos,
        OffsetIni := #NumBytes,
        Valor     := #Valor,
        OffsetFin := #Offset
      );  // Llamo a ObtenerStrinAtributo

      L     #Offset;
      SLD   3;
      LAR2;  // Recupero que offset tiene la String

// --- Ya esta convertido el Valor a ASCI - Fin Peso
Peso_NUUT_EventoUT:NOP   0;


////////////////////////////////////////////////////////////////////////////////
// --- Atributo de ANCHURA COTA (Si es necesario) ---
      SET;
      AN    "DB850_DefinicionMesas".Mesa[#NumMesa].AtributosGalibo_DeEvento.Cota_Anchura;  // Tiene Cota de Anchura ?
      JC    CotaAnchura_NUUT_EventoUT;

      L     "DB815_UTs_Datos".UT[#NumeroUT].CotaAnchura;
      T     #Valor;

      OPN   DB [#DBEventos];
      L     '[';  // Evento - Atributo Anchura Cota '[COTW]'
      T     DBB [AR2, P#0.0];
      L     'COTW';
      T     DBD [AR2, P#1.0];
      L     ']';
      T     DBB [AR2, P#5.0];
      +AR2  P#6.0;

// --- Convertir Valor a ASCII -  Anchura Cota
      TAR2;
      SRD   3;
      T     #NumBytes;  // Miro que offset tiene la String

      CALL  "FC893_Obtener_StringDelAtributo"
      ( DB_String := #NumDBEventos,
        OffsetIni := #NumBytes,
        Valor     := #Valor,
        OffsetFin := #Offset
      );  // Llamo a ObtenerStrinAtributo

      L     #Offset;
      SLD   3;
      LAR2;  // Recupero que offset tiene la String

// --- Ya esta convertido el Valor a ASCI - Fin Anchura Cota
CotaAnchura_NUUT_EventoUT:NOP   0;


////////////////////////////////////////////////////////////////////////////////
// --- Atributo de LARGURA COTA (Si es necesario) ---
      SET;
      AN    "DB850_DefinicionMesas".Mesa[#NumMesa].AtributosGalibo_DeEvento.Cota_Profundidad;  // Tiene Cota de Profundidad ?
      JC    CotaLargura_NUUT_EventoUT;

      L     "DB815_UTs_Datos".UT[#NumeroUT].CotaProfundidad;
      T     #Valor;

      OPN   DB [#DBEventos];
      L     '[';  // Evento - Atributo Largura Cota '[COTL]'
      T     DBB [AR2, P#0.0];
      L     'COTL';
      T     DBD [AR2, P#1.0];
      L     ']';
      T     DBB [AR2, P#5.0];
      +AR2  P#6.0;

// --- Convertir Valor a ASCII -  Largura Cota
      TAR2;
      SRD   3;
      T     #NumBytes;  // Miro que offset tiene la String

      CALL  "FC893_Obtener_StringDelAtributo"
      ( DB_String := #NumDBEventos,
        OffsetIni := #NumBytes,
        Valor     := #Valor,
        OffsetFin := #Offset
      );  // Llamo a ObtenerStrinAtributo

      L     #Offset;
      SLD   3;
      LAR2;  // Recupero que offset tiene la String

// --- Ya esta convertido el Valor a ASCI - Fin Largura Cota
CotaLargura_NUUT_EventoUT:NOP   0;


////////////////////////////////////////////////////////////////////////////////
////////////////////////////////////////////////////////////////////////////////
////////////////////////////////////////////////////////////////////////////////
////////////////////////////////////////////////////////////////////////////////
// --- Atributo de TIPO, HUECO y TACO (Si es necesario) ---
      SET;  // Tiene Taco ?
      AN    "DB850_DefinicionMesas".Mesa[#NumMesa].AtributosGalibo_DeEvento.Taco;
      JC    CodigoTaco_NUUT_EventosUT;

      OPN   DB [#DBEventos];
      L     '[';  // Evento - Atributo Galibo Taco '[TACO]'
      T     DBB [AR2, P#0.0];
      L     'TACO';
      T     DBD [AR2, P#1.0];
      L     ']';
      T     DBB [AR2, P#5.0];
      +AR2  P#6.0;

      L     "DB815_UTs_Datos".UT[#NumeroUT].GaliboTaco;
      T     #Valor;

// --- Convertir Valor a ASCII -  Taco
      TAR2;
      SRD   3;
      T     #NumBytes;  // Miro que offset tiene la String

      CALL  "FC893_Obtener_StringDelAtributo"
      ( DB_String := #NumDBEventos,
        OffsetIni := #NumBytes,
        Valor     := #Valor,
        OffsetFin := #Offset
      );  // Llamo a ObtenerStrinAtributo

      L     #Offset;
      SLD   3;
      LAR2;  // Recupero que offset tiene la String

// --- Ya esta convertido el Valor a ASCI - Fin Taco
CodigoTaco_NUUT_EventosUT:NOP   0;


////////////////////////////////////////////////////////////////////////////////
      SET;  // Tiene Hueco ?
      AN    "DB850_DefinicionMesas".Mesa[#NumMesa].AtributosGalibo_DeEvento.Hueco;
      JC    CodigoHueco_NUUT_EventosUT;

      OPN   DB [#DBEventos];
      L     '[';  // Evento - Atributo Galibo Hueco '[HUEC]'
      T     DBB [AR2, P#0.0];
      L     'HUEC';
      T     DBD [AR2, P#1.0];
      L     ']';
      T     DBB [AR2, P#5.0];
      +AR2  P#6.0;

      L     "DB815_UTs_Datos".UT[#NumeroUT].GaliboHueco;
      T     #Valor;

// --- Convertir Valor a ASCII -  Hueco
      TAR2;
      SRD   3;
      T     #NumBytes;  // Miro que offset tiene la String

      CALL  "FC893_Obtener_StringDelAtributo"
      ( DB_String := #NumDBEventos,
        OffsetIni := #NumBytes,
        Valor     := #Valor,
        OffsetFin := #Offset
      );  // Llamo a ObtenerStrinAtributo

      L     #Offset;
      SLD   3;
      LAR2;  // Recupero que offset tiene la String

// --- Ya esta convertido el Valor a ASCI - Fin Hueco
CodigoHueco_NUUT_EventosUT:NOP   0;


////////////////////////////////////////////////////////////////////////////////
      SET;  // Tiene Hueco R ?
      AN    "DB850_DefinicionMesas".Mesa[#NumMesa].AtributosGalibo_DeEvento.HuecoRemontado;
      JC    CodigoHuecoR_NUUT_EventosUT;

      OPN   DB [#DBEventos];
      L     '[';  // Evento - Atributo Galibo Hueco '[HUEC]'
      T     DBB [AR2, P#0.0];
      L     'HUER';
      T     DBD [AR2, P#1.0];
      L     ']';
      T     DBB [AR2, P#5.0];
      +AR2  P#6.0;

      L     "DB815_UTs_Datos".UT[#NumeroUT].GaliboHuecoRemontado;
      T     #Valor;

// --- Convertir Valor a ASCII -  Huer
      TAR2;
      SRD   3;
      T     #NumBytes;  // Miro que offset tiene la String

      CALL  "FC893_Obtener_StringDelAtributo"
      ( DB_String := #NumDBEventos,
        OffsetIni := #NumBytes,
        Valor     := #Valor,
        OffsetFin := #Offset
      );  // Llamo a ObtenerStrinAtributo

      L     #Offset;
      SLD   3;
      LAR2;  // Recupero que offset tiene la String

// --- Ya esta convertido el Valor a ASCI - Fin Huer
CodigoHuecoR_NUUT_EventosUT:NOP   0;


////////////////////////////////////////////////////////////////////////////////
      SET;  // Tiene Tipo ?
      AN    "DB850_DefinicionMesas".Mesa[#NumMesa].AtributosGalibo_DeEvento.Tipo;
      JC    CodigoTipo_NUUT_EventosUT;

      OPN   DB [#DBEventos];
      L     '[';  // Evento - Atributo Galibo Hueco '[HUEC]'
      T     DBB [AR2, P#0.0];
      L     'TIPO';
      T     DBD [AR2, P#1.0];
      L     ']';
      T     DBB [AR2, P#5.0];
      +AR2  P#6.0;

      L     "DB815_UTs_Datos".UT[#NumeroUT].GaliboTipoCarga;
      L     W#16#F;
      <>I;
      JC    CodigoTipoExiste_NUUT_EventosUT;

      OPN   DB [#DBEventos];
      L     'ERRO';
      T     DBD [AR2, P#0.0];
      +AR2  P#4.0;

      JU    CodigoTipo_NUUT_EventosUT;

CodigoTipoExiste_NUUT_EventosUT:NOP   0;
      L     "DB815_UTs_Datos".UT[#NumeroUT].GaliboTipoCarga;
      L     3000;
      +I;
      T     #Convertir;
      CALL  "FC895_Obtener_EtiquetaDeValor"
      ( ValorEvento    := #Convertir,
        EtiquetaEvento := #Conversion
      );

      OPN   DB [#DBEventos];
      L     #Conversion;
      T     DBD [AR2, P#0.0];
      +AR2  P#4.0;

CodigoTipo_NUUT_EventosUT:NOP   0;

////////////////////////////////////////////////////////////////////////////////
////////////////////////////////////////////////////////////////////////////////
////////////////////////////////////////////////////////////////////////////////
////////////////////////////////////////////////////////////////////////////////


////////////////////////////////////////////////////////////////////////////////
////////////////////////////////////////////////////////////////////////////////
////////////////////////////////////////////////////////////////////////////////
////////////////////////////////////////////////////////////////////////////////
// --- Atributo de COLOR (Si es necesario) ---
      SET;  // Tiene Color ?
      AN    "DB850_DefinicionMesas".Mesa[#NumMesa].AtributosGalibo_DeEvento.Color;
      JC    CodigoColor_NUUT_EventosUT;

      OPN   DB [#DBEventos];
      L     '[';  // Evento - Atributo Galibo Hueco '[HUEC]'
      T     DBB [AR2, P#0.0];
      L     'COLO';
      T     DBD [AR2, P#1.0];
      L     ']';
      T     DBB [AR2, P#5.0];
      +AR2  P#6.0;

      L     "DB815_UTs_Datos".UT[#NumeroUT].GaliboColor;
      L     W#16#F;
      <>I;
      JC    CodigoColorExiste_NUUT_EventosUT;

      OPN   DB [#DBEventos];
      L     'ERRO';  // ERROR De COLOR
      T     DBD [AR2, P#0.0];
      +AR2  P#4.0;

      JU    CodigoColor_NUUT_EventosUT;

CodigoColorExiste_NUUT_EventosUT:NOP   0;
      L     "DB815_UTs_Datos".UT[#NumeroUT].GaliboColor;
      L     3100;
      +I;
      T     #Convertir;
      CALL  "FC895_Obtener_EtiquetaDeValor"
      ( ValorEvento    := #Convertir,
        EtiquetaEvento := #Conversion
      );

      OPN   DB [#DBEventos];
      L     #Conversion;
      T     DBD [AR2, P#0.0];
      +AR2  P#4.0;

CodigoColor_NUUT_EventosUT:NOP   0;


////////////////////////////////////////////////////////////////////////////////
      SET;
      AN    "DB850_DefinicionMesas".Mesa[#NumMesa].AtributosGalibo_DeEvento.Patin;
      JC    CodigoPatin_NUUT_EventosUT;  // Tiene Patin ?

      OPN   DB [#DBEventos];
      L     '[';  // Evento - Atributo Galibo Patin '[PATI]'
      T     DBB [AR2, P#0.0];
      L     'PATI';
      T     DBD [AR2, P#1.0];
      L     ']';
      T     DBB [AR2, P#5.0];
      +AR2  P#6.0;

      L     "DB815_UTs_Datos".UT[#NumeroUT].GaliboPatin;
      T     #Valor;

// --- Convertir Valor a ASCII -  Patin
      TAR2;
      SRD   3;
      T     #NumBytes;  // Miro que offset tiene la String

      CALL  "FC893_Obtener_StringDelAtributo"
      ( DB_String := #NumDBEventos,
        OffsetIni := #NumBytes,
        Valor     := #Valor,
        OffsetFin := #Offset
      );  // Llamo a ObtenerStrinAtributo

      L     #Offset;
      SLD   3;
      LAR2;  // Recupero que offset tiene la String

// --- Ya esta convertido el Valor a ASCI - Fin Patin
CodigoPatin_NUUT_EventosUT:NOP   0;





////////////////////////////////////////////////////////////////////////////////
// --- Atributo de ETIQUETA (Si es necesario) --- Router
      SET;  // Tiene Etiqueta
      AN    "DB850_DefinicionMesas".Mesa[#NumMesa].AtributosGalibo_DeEvento.EtiquetaRouter;
      JC    FinEtiquetaRouter_NUUT_EventoUT;

      OPN   DB [#DBEventos];
      L     '[';  // Evento - Atributo Etiqueta '[SSCC]'
      T     DBB [AR2, P#0.0];
      L     'SSCC';
      T     DBD [AR2, P#1.0];
      L     ']';
      T     DBB [AR2, P#5.0];
      +AR2  P#6.0;

      L     "DB814_UTs_Etiqueta".UT[#NumeroUT].EtiquetaRouter;
      T     #Valor;

// --- Convertir Valor a ASCII -  Etiqueta de Router
      TAR2;
      SRD   3;
      T     #NumBytes;  // Miro que offset tiene la String

      CALL  "FC893_Obtener_StringDelAtributo"
      ( DB_String := #NumDBEventos,
        OffsetIni := #NumBytes,
        Valor     := #Valor,
        OffsetFin := #Offset
      );  // Llamo a ObtenerStrinAtributo

      L     #Offset;
      SLD   3;
      LAR2;  // Recupero que offset tiene la String

// --- Ya esta convertido el Valor a ASCI - Fin Etiqueta de Router
FinEtiquetaRouter_NUUT_EventoUT:NOP   0;





////////////////////////////////////////////////////////////////////////////////
// --- Atributo de ETIQUETA (Si es necesario) ---  STRING
      SET;  // Tiene Etiqueta
      AN    "DB850_DefinicionMesas".Mesa[#NumMesa].AtributosGalibo_DeEvento.EtiquetaString;
      JC    FinEtiquetaString_NUUT_EventoUT;

      OPN   DB [#DBEventos];
      L     '[';  // Evento - Atributo Etiqueta '[SSCC]'
      T     DBB [AR2, P#0.0];
      L     'SSCC';
      T     DBD [AR2, P#1.0];
      L     ']';
      T     DBB [AR2, P#5.0];
      +AR2  P#6.0;

      L     2;  // Puntero a la Etiqueta
      T     #IndiceEtiqueta;

BucleEtiquetastring_NUUT_EventoUT:NOP   0;
      L     "DB814_UTs_Etiqueta".UT[#NumeroUT].Etiqueta[#IndiceEtiqueta];
      T     #Valor;  // Recoge el caracter de la Etiqueta

      L     #Valor;
      L     0;
      ==D;  // Es Final de Etiqueta?
      JC    FinEtiquetaString_NUUT_EventoUT;

      OPN   DB [#DBEventos];
      L     #Valor;
      T     DBB [AR2, P#0.0];

      L     #IndiceEtiqueta;  // Siguiente Caracter
      L     1;
      +I;
      T     #IndiceEtiqueta;
      +AR2  P#1.0;

      JU    BucleEtiquetastring_NUUT_EventoUT;

FinEtiquetaString_NUUT_EventoUT:NOP   0;


////////////////////////////////////////////////////////////////////////////////-
// --- Final del Formato del Evento ---

      OPN   DB [#DBEventos];  // DB de Eventos Generados (A Emitir)
      L     '}';  // Fin de Evento '}'
      T     DBB [AR2, P#0.0];
      +AR2  P#1.0;

////////////////////////////////////////////////////////////////////////////////
////////////////////////////////////////////////////////////////////////////////
////////////////////////////////////////////////////////////////////////////////
////////////////////////////////////////////////////////////////////////////////
// Dar por formateado el Evento
// Borrar la UT de la Base de datos (Por Presencias Multiples de las Mesas)
// Solo no se borra cuando la Mesa es Remota, no debe ni entrar aqui.

      CALL  "FC722_EliminarUT_DeMesa"
      ( NumeroUT := #NumeroUT
      );

      JU    FinBucles_EventosUT;

// Fin del Evento NUUT
////////////////////////////////////////////////////////////////////////////////
////////////////////////////////////////////////////////////////////////////////
////////////////////////////////////////////////////////////////////////////////
////////////////////////////////////////////////////////////////////////////////



NETWORK
TITLE = ---- Evento de UT - Refresco de Datos de la UT -- DATO
GenerarEvento_DATO_EventoUT:NOP   0;

////////////////////////////////////////////////////////////////////////////////
////////////////////////////////////////////////////////////////////////////////
////////////////////////////////////////////////////////////////////////////////
////////////////////////////////////////////////////////////////////////////////
// -- Formateo del Evento DATO - Refresco de Datos de la UT

      L     #P_Eventos;
      LAR2;  // Puntero al DB de Eventos Generados

      TAR2;  // Mirar si es el primer evento de la lista
      L     0;
      ==I;
      JC    InicioBuffer_DATO_EventosUT;  // Es el primero

      OPN   DB [#DBEventos];  // Hay que añadir si no es el primer evento
      L     ',';  // Separador entre eventos ','
      T     DBB [AR2, P#0.0];
      +AR2  P#1.0;

InicioBuffer_DATO_EventosUT:NOP   0;
      OPN   DB [#DBEventos];  // DB de Eventos Generados (A Emitir)
      L     '{';  // Inicio de Evento '{'
      T     DBB [AR2, P#0.0];
      +AR2  P#1.0;

      L     'DATO';  // Evento 'DATO'
      T     DBD [AR2, P#0.0];
      +AR2  P#4.0;


////////////////////////////////////////////////////////////////////////////////
      L     '[';  // Evento - Atributo Mckey '[MCKY]'
      T     DBB [AR2, P#0.0];
      L     'MCKY';
      T     DBD [AR2, P#1.0];
      L     ']';
      T     DBB [AR2, P#5.0];
      +AR2  P#6.0;

      L     "DB812_UTs_Control".UT[#NumeroUT].Mckey;
      T     #Valor;

// --- Convertir Valor a ASCII - Mckey
      TAR2;
      SRD   3;
      T     #NumBytes;  // Miro que offset tiene la String

      CALL  "FC893_Obtener_StringDelAtributo"
      ( DB_String := #NumDBEventos,
        OffsetIni := #NumBytes,
        Valor     := #Valor,
        OffsetFin := #Offset
      );  // Llamo a ObtenerStrinAtributo

      L     #Offset;
      SLD   3;
      LAR2;  // Recupero que offset tiene la String

// --- Ya esta convertido el Valor a ASCI - Fin Mckey


////////////////////////////////////////////////////////////////////////////////
      OPN   DB [#DBEventos];
      L     '[';  // Evento - Atributo Mesa Actual '[MESA]'
      T     DBB [AR2, P#0.0];
      L     'MESA';
      T     DBD [AR2, P#1.0];
      L     ']';
      T     DBB [AR2, P#5.0];
      +AR2  P#6.0;

      L     "DB812_UTs_Control".UT[#NumeroUT].MesaActual;
      T     #Valor;

// --- Convertir Valor a ASCII -  Mesa Actual
      TAR2;
      SRD   3;
      T     #NumBytes;  // Miro que offset tiene la String

      CALL  "FC893_Obtener_StringDelAtributo"
      ( DB_String := #NumDBEventos,
        OffsetIni := #NumBytes,
        Valor     := #Valor,
        OffsetFin := #Offset
      );  // Llamo a ObtenerStrinAtributo

      L     #Offset;
      SLD   3;
      LAR2;  // Recupero que offset tiene la String

// --- Ya esta convertido el Valor a ASCI - Fin Mesa Actual


////////////////////////////////////////////////////////////////////////////////
////////////////////////////////////////////////////////////////////////////////
////////////////////////////////////////////////////////////////////////////////
////////////////////////////////////////////////////////////////////////////////
// --- Caracteristicas de la UT a Emitir


////////////////////////////////////////////////////////////////////////////////
// --- Atributo de ALTURA COTA (Si es necesario) ---
      SET;  // Tiene Cota de Altura ?
      AN    "DB850_DefinicionMesas".Mesa[#NumMesa].AtributosGalibo_DeEvento.Cota_Altura;
      JC    CotaAltura_DATO_EventoUT;

      L     "DB815_UTs_Datos".UT[#NumeroUT].CotaAltura;
      T     #Valor;

      OPN   DB [#DBEventos];
      L     '[';  // Evento - Atributo Altura Cota '[COTA]'
      T     DBB [AR2, P#0.0];
      L     'COTA';
      T     DBD [AR2, P#1.0];
      L     ']';
      T     DBB [AR2, P#5.0];
      +AR2  P#6.0;

// --- Convertir Valor a ASCII -  Altura Cota
      TAR2;
      SRD   3;
      T     #NumBytes;  // Miro que offset tiene la String

      CALL  "FC893_Obtener_StringDelAtributo"
      ( DB_String := #NumDBEventos,
        OffsetIni := #NumBytes,
        Valor     := #Valor,
        OffsetFin := #Offset
      );  // Llamo a ObtenerStrinAtributo

      L     #Offset;
      SLD   3;
      LAR2;  // Recupero que offset tiene la String

// --- Ya esta convertido el Valor a ASCI - Fin Altura Cota
CotaAltura_DATO_EventoUT:NOP   0;


////////////////////////////////////////////////////////////////////////////////
////////////////////////////////////////////////////////////////////////////////
////////////////////////////////////////////////////////////////////////////////
////////////////////////////////////////////////////////////////////////////////
// --- Atributo de GALIBO (Si es necesario) ---
      SET;  // Tiene Altura ?
      AN    "DB850_DefinicionMesas".Mesa[#NumMesa].AtributosGalibo_DeEvento.Altura;
      JC    CodigoAltura_DATO_EventoUT;

      OPN   DB [#DBEventos];
      L     '[';  // Evento - Atributo Galibo Altura '[ALTO]'
      T     DBB [AR2, P#0.0];
      L     'ALTO';
      T     DBD [AR2, P#1.0];
      L     ']';
      T     DBB [AR2, P#5.0];
      +AR2  P#6.0;

      L     "DB815_UTs_Datos".UT[#NumeroUT].GaliboAltura;
      T     #Valor;

// --- Convertir Valor a ASCII -  Alto
      TAR2;
      SRD   3;
      T     #NumBytes;  // Miro que offset tiene la String

      CALL  "FC893_Obtener_StringDelAtributo"
      ( DB_String := #NumDBEventos,
        OffsetIni := #NumBytes,
        Valor     := #Valor,
        OffsetFin := #Offset
      );  // Llamo a ObtenerStrinAtributo

      L     #Offset;
      SLD   3;
      LAR2;  // Recupero que offset tiene la String


// nieves inicio modificación emisión atributo VACI

//Comprobar si tenemos que emitir el evento

      SET;
      L     "DB815_UTs_Datos".UT[#NumeroUT].GaliboVacia;
      L     0;
      ==I;
      JC    CodigoAltura_DATO_EventoUT;

      OPN   DB [#DBEventos];
      L     '[';  // Evento - Atributo Galibo Altura '[ALTO]'
      T     DBB [AR2, P#0.0];
      L     'VACI';
      T     DBD [AR2, P#1.0];
      L     ']';
      T     DBB [AR2, P#5.0];
      +AR2  P#6.0;

      L     "DB815_UTs_Datos".UT[#NumeroUT].GaliboVacia;
      L     1;
      -I;
      T     #Valor;

// --- Convertir Valor a ASCII -  VACIO
      TAR2;
      SRD   3;
      T     #NumBytes;  // Miro que offset tiene la String

      CALL  "FC893_Obtener_StringDelAtributo"
      ( DB_String := #NumDBEventos,
        OffsetIni := #NumBytes,
        Valor     := #Valor,
        OffsetFin := #Offset
      );  // Llamo a ObtenerStrinAtributo


      L     #Offset;
      SLD   3;
      LAR2;  // Recupero que offset tiene la String


// fin modificación atributo VACI

// --- Ya esta convertido el Valor a ASCI - Fin Alto
CodigoAltura_DATO_EventoUT:NOP   0;


////////////////////////////////////////////////////////////////////////////////
      SET;  // Tien Anchura ?
      AN    "DB850_DefinicionMesas".Mesa[#NumMesa].AtributosGalibo_DeEvento.Anchura;
      JC    CodigAnchura_DATO_EventoUT;

      OPN   DB [#DBEventos];
      L     '[';  // Evento - Atributo Galibo Anchura '[ANCH]'
      T     DBB [AR2, P#0.0];
      L     'ANCH';
      T     DBD [AR2, P#1.0];
      L     ']';
      T     DBB [AR2, P#5.0];
      +AR2  P#6.0;

      L     "DB815_UTs_Datos".UT[#NumeroUT].GaliboAnchura;
      T     #Valor;

// --- Convertir Valor a ASCII -  Anchura
      TAR2;
      SRD   3;
      T     #NumBytes;  // Miro que offset tiene la String

      CALL  "FC893_Obtener_StringDelAtributo"
      ( DB_String := #NumDBEventos,
        OffsetIni := #NumBytes,
        Valor     := #Valor,
        OffsetFin := #Offset
      );  // Llamo a ObtenerStrinAtributo

      L     #Offset;
      SLD   3;
      LAR2;  // Recupero que offset tiene la String

// --- Ya esta convertido el Valor a ASCI - Fin Anchura
CodigAnchura_DATO_EventoUT:NOP   0;


////////////////////////////////////////////////////////////////////////////////
      SET;  // Tiene Profundidad ?
      AN    "DB850_DefinicionMesas".Mesa[#NumMesa].AtributosGalibo_DeEvento.Profundidad;
      JC    CodigLargura_DATO_EventoUT;

      OPN   DB [#DBEventos];
      L     '[';  // Evento - Atributo Galibo Profuncidad '[PROF]'
      T     DBB [AR2, P#0.0];
      L     'PROF';
      T     DBD [AR2, P#1.0];
      L     ']';
      T     DBB [AR2, P#5.0];
      +AR2  P#6.0;

      L     "DB815_UTs_Datos".UT[#NumeroUT].GaliboProfundidad;
      T     #Valor;

// --- Convertir Valor a ASCII -  Largura
      TAR2;
      SRD   3;
      T     #NumBytes;  // Miro que offset tiene la String

      CALL  "FC893_Obtener_StringDelAtributo"
      ( DB_String := #NumDBEventos,
        OffsetIni := #NumBytes,
        Valor     := #Valor,
        OffsetFin := #Offset
      );  // Llamo a ObtenerStrinAtributo

      L     #Offset;
      SLD   3;
      LAR2;  // Recupero que offset tiene la String

// --- Ya esta convertido el Valor a ASCI - Fin Largura
CodigLargura_DATO_EventoUT:NOP   0;


////////////////////////////////////////////////////////////////////////////////
      SET;  // Tiene Remontado ?
      AN    "DB850_DefinicionMesas".Mesa[#NumMesa].AtributosGalibo_DeEvento.Remontado;
      JC    CodigRemontado_DATO_EventoUT;

      OPN   DB [#DBEventos];
      L     '[';  // Evento - Atributo Galibo Remontada '[REMO]'
      T     DBB [AR2, P#0.0];
      L     'REMO';
      T     DBD [AR2, P#1.0];
      L     ']';
      T     DBB [AR2, P#5.0];
      +AR2  P#6.0;

      L     "DB815_UTs_Datos".UT[#NumeroUT].GaliboRemontada;
      L     1;
      -I;
      L     W#16#30;
      +I;
      OPN   DB [#DBEventos];
      T     DBB [AR2, P#0.0];
      +AR2  P#1.0;

CodigRemontado_DATO_EventoUT:NOP   0;


////////////////////////////////////////////////////////////////////////////////
// --- Atributo de PESO (Si es necesario) ---
      SET;  // Tiene Peso ?
      AN    "DB850_DefinicionMesas".Mesa[#NumMesa].AtributosGalibo_DeEvento.Peso;
      JC    Peso_DATO_EventoUT;

      OPN   DB [#DBEventos];
      L     '[';  // Evento - Atributo Peso '[PESO]'
      T     DBB [AR2, P#0.0];
      L     'PESO';
      T     DBD [AR2, P#1.0];
      L     ']';
      T     DBB [AR2, P#5.0];
      +AR2  P#6.0;

      L     "DB815_UTs_Datos".UT[#NumeroUT].Peso;
      T     #Valor;

// --- Convertir Valor a ASCII -  Peso
      TAR2;
      SRD   3;
      T     #NumBytes;  // Miro que offset tiene la String

      CALL  "FC893_Obtener_StringDelAtributo"
      ( DB_String := #NumDBEventos,
        OffsetIni := #NumBytes,
        Valor     := #Valor,
        OffsetFin := #Offset
      );  // Llamo a ObtenerStrinAtributo

      L     #Offset;
      SLD   3;
      LAR2;  // Recupero que offset tiene la String

// --- Ya esta convertido el Valor a ASCI - Fin Peso
Peso_DATO_EventoUT:NOP   0;


////////////////////////////////////////////////////////////////////////////////
// --- Atributo de ANCHURA COTA (Si es necesario) ---
      SET;  // Tiene Cota de Anchura ?
      AN    "DB850_DefinicionMesas".Mesa[#NumMesa].AtributosGalibo_DeEvento.Cota_Anchura;
      JC    CotaAnchura_DATO_EventoUT;

      L     "DB815_UTs_Datos".UT[#NumeroUT].CotaAnchura;
      T     #Valor;

      OPN   DB [#DBEventos];
      L     '[';  // Evento - Atributo Anchura Cota '[COTW]'
      T     DBB [AR2, P#0.0];
      L     'COTW';
      T     DBD [AR2, P#1.0];
      L     ']';
      T     DBB [AR2, P#5.0];
      +AR2  P#6.0;

// --- Convertir Valor a ASCII -  Anchura Cota
      TAR2;
      SRD   3;
      T     #NumBytes;  // Miro que offset tiene la String

      CALL  "FC893_Obtener_StringDelAtributo"
      ( DB_String := #NumDBEventos,
        OffsetIni := #NumBytes,
        Valor     := #Valor,
        OffsetFin := #Offset
      );  // Llamo a ObtenerStrinAtributo

      L     #Offset;
      SLD   3;
      LAR2;  // Recupero que offset tiene la String

// --- Ya esta convertido el Valor a ASCI - Fin Anchura Cota
CotaAnchura_DATO_EventoUT:NOP   0;


////////////////////////////////////////////////////////////////////////////////
// --- Atributo de LARGURA COTA (Si es necesario) ---
      SET;  // Tiene Cota de Profundidad ?
      AN    "DB850_DefinicionMesas".Mesa[#NumMesa].AtributosGalibo_DeEvento.Cota_Profundidad;
      JC    CotaLargura_DATO_EventoUT;

      L     "DB815_UTs_Datos".UT[#NumeroUT].CotaProfundidad;
      T     #Valor;

      OPN   DB [#DBEventos];
      L     '[';  // Evento - Atributo Largura Cota '[COTL]'
      T     DBB [AR2, P#0.0];
      L     'COTL';
      T     DBD [AR2, P#1.0];
      L     ']';
      T     DBB [AR2, P#5.0];
      +AR2  P#6.0;

// --- Convertir Valor a ASCII -  Largura Cota
      TAR2;
      SRD   3;
      T     #NumBytes;  // Miro que offset tiene la String

      CALL  "FC893_Obtener_StringDelAtributo"
      ( DB_String := #NumDBEventos,
        OffsetIni := #NumBytes,
        Valor     := #Valor,
        OffsetFin := #Offset
      );  // Llamo a ObtenerStrinAtributo

      L     #Offset;
      SLD   3;
      LAR2;  // Recupero que offset tiene la String

// --- Ya esta convertido el Valor a ASCI - Fin Largura Cota
CotaLargura_DATO_EventoUT:NOP   0;


////////////////////////////////////////////////////////////////////////////////
////////////////////////////////////////////////////////////////////////////////
////////////////////////////////////////////////////////////////////////////////
// --- Atributo de TIPO, HUECO y TACO (Si es necesario) ---
      SET;  // Tiene Taco ?
      AN    "DB850_DefinicionMesas".Mesa[#NumMesa].AtributosGalibo_DeEvento.Taco;
      JC    CodigoTaco_DATO_EventoUT;

      OPN   DB [#DBEventos];
      L     '[';  // Evento - Atributo Galibo Taco '[TACO]'
      T     DBB [AR2, P#0.0];
      L     'TACO';
      T     DBD [AR2, P#1.0];
      L     ']';
      T     DBB [AR2, P#5.0];
      +AR2  P#6.0;

      L     "DB815_UTs_Datos".UT[#NumeroUT].GaliboTaco;
      T     #Valor;

// --- Convertir Valor a ASCII -  Taco
      TAR2;
      SRD   3;
      T     #NumBytes;  // Miro que offset tiene la String

      CALL  "FC893_Obtener_StringDelAtributo"
      ( DB_String := #NumDBEventos,
        OffsetIni := #NumBytes,
        Valor     := #Valor,
        OffsetFin := #Offset
      );  // Llamo a ObtenerStrinAtributo

      L     #Offset;
      SLD   3;
      LAR2;  // Recupero que offset tiene la String

// --- Ya esta convertido el Valor a ASCI - Fin Taco
CodigoTaco_DATO_EventoUT:NOP   0;


////////////////////////////////////////////////////////////////////////////////
      SET;  // Tiene Hueco ?
      AN    "DB850_DefinicionMesas".Mesa[#NumMesa].AtributosGalibo_DeEvento.Hueco;
      JC    CodigoHueco_DATO_EventoUT;

      OPN   DB [#DBEventos];
      L     '[';  // Evento - Atributo Galibo Hueco '[HUEC]'
      T     DBB [AR2, P#0.0];
      L     'HUEC';
      T     DBD [AR2, P#1.0];
      L     ']';
      T     DBB [AR2, P#5.0];
      +AR2  P#6.0;

      L     "DB815_UTs_Datos".UT[#NumeroUT].GaliboHueco;
      T     #Valor;

// --- Convertir Valor a ASCII -  Hueco
      TAR2;
      SRD   3;
      T     #NumBytes;  // Miro que offset tiene la String

      CALL  "FC893_Obtener_StringDelAtributo"
      ( DB_String := #NumDBEventos,
        OffsetIni := #NumBytes,
        Valor     := #Valor,
        OffsetFin := #Offset
      );  // Llamo a ObtenerStrinAtributo

      L     #Offset;
      SLD   3;
      LAR2;  // Recupero que offset tiene la String

// --- Ya esta convertido el Valor a ASCI - Fin Hueco
CodigoHueco_DATO_EventoUT:NOP   0;


////////////////////////////////////////////////////////////////////////////////
      SET;  // Tiene Hueco_R
      AN    "DB850_DefinicionMesas".Mesa[#NumMesa].AtributosGalibo_DeEvento.HuecoRemontado;
      JC    CodigoHuecoR_DATO_EventoUT;

      OPN   DB [#DBEventos];
      L     '[';  // Evento - Atributo Galibo Hueco '[HUEC]'
      T     DBB [AR2, P#0.0];
      L     'HUER';
      T     DBD [AR2, P#1.0];
      L     ']';
      T     DBB [AR2, P#5.0];
      +AR2  P#6.0;

      L     "DB815_UTs_Datos".UT[#NumeroUT].GaliboHuecoRemontado;
      T     #Valor;

// --- Convertir Valor a ASCII -  Hueco R
      TAR2;
      SRD   3;
      T     #NumBytes;  // Miro que offset tiene la String

      CALL  "FC893_Obtener_StringDelAtributo"
      ( DB_String := #NumDBEventos,
        OffsetIni := #NumBytes,
        Valor     := #Valor,
        OffsetFin := #Offset
      );  // Llamo a ObtenerStrinAtributo

      L     #Offset;
      SLD   3;
      LAR2;  // Recupero que offset tiene la String

// --- Ya esta convertido el Valor a ASCI - Fin Hueco R
CodigoHuecoR_DATO_EventoUT:NOP   0;


////////////////////////////////////////////////////////////////////////////////
      SET;  // Tiene Tipo ?
      AN    "DB850_DefinicionMesas".Mesa[#NumMesa].AtributosGalibo_DeEvento.Tipo;
      JC    CodigoTipo_DATO_EventoUT;

      OPN   DB [#DBEventos];
      L     '[';  // Evento - Atributo Galibo Hueco '[HUEC]'
      T     DBB [AR2, P#0.0];
      L     'TIPO';
      T     DBD [AR2, P#1.0];
      L     ']';
      T     DBB [AR2, P#5.0];
      +AR2  P#6.0;

      L     "DB815_UTs_Datos".UT[#NumeroUT].GaliboTipoCarga;
      L     W#16#F;
      <>I;
      JC    CodigoTipoExiste_DATO_EventoUT;

      OPN   DB [#DBEventos];
      L     'ERRO';
      T     DBD [AR2, P#0.0];
      +AR2  P#4.0;

      JU    CodigoTipo_DATO_EventoUT;

CodigoTipoExiste_DATO_EventoUT:NOP   0;
      L     "DB815_UTs_Datos".UT[#NumeroUT].GaliboTipoCarga;
      L     3000;
      +I;
      T     #Convertir;
      CALL  "FC895_Obtener_EtiquetaDeValor"
      ( ValorEvento    := #Convertir,
        EtiquetaEvento := #Conversion
      );

      OPN   DB [#DBEventos];
      L     #Conversion;
      T     DBD [AR2, P#0.0];
      +AR2  P#4.0;

CodigoTipo_DATO_EventoUT:NOP   0;


////////////////////////////////////////////////////////////////////////////////
////////////////////////////////////////////////////////////////////////////////
////////////////////////////////////////////////////////////////////////////////
// --- Atributo de COLOR (Si es necesario) ---
      SET;  // Tiene Color ?
      AN    "DB850_DefinicionMesas".Mesa[#NumMesa].AtributosGalibo_DeEvento.Color;
      JC    CodigoColor_DATO_EventoUT;

      OPN   DB [#DBEventos];
      L     '[';  // Evento - Atributo Galibo Hueco '[HUEC]'
      T     DBB [AR2, P#0.0];
      L     'COLO';
      T     DBD [AR2, P#1.0];
      L     ']';
      T     DBB [AR2, P#5.0];
      +AR2  P#6.0;

      L     "DB815_UTs_Datos".UT[#NumeroUT].GaliboColor;
      L     W#16#F;
      <>I;
      JC    CodigoColorExiste_DATO_EventoUT;

      OPN   DB [#DBEventos];
      L     'ERRO';
      T     DBD [AR2, P#0.0];
      +AR2  P#4.0;

      JU    CodigoColor_DATO_EventoUT;

CodigoColorExiste_DATO_EventoUT:NOP   0;
      L     "DB815_UTs_Datos".UT[#NumeroUT].GaliboColor;
      L     3100;
      +I;
      T     #Convertir;
      CALL  "FC895_Obtener_EtiquetaDeValor"
      ( ValorEvento    := #Convertir,
        EtiquetaEvento := #Conversion
      );

      OPN   DB [#DBEventos];
      L     #Conversion;
      T     DBD [AR2, P#0.0];
      +AR2  P#4.0;

CodigoColor_DATO_EventoUT:NOP   0;

////////////////////////////////////////////////////////////////////////////////
      SET;  // Tiene Patin ?
      AN    "DB850_DefinicionMesas".Mesa[#NumMesa].AtributosGalibo_DeEvento.Patin;
      JC    CodigoPatin_DATO_EventoUT;

      OPN   DB [#DBEventos];
      L     '[';  // Evento - Atributo Galibo Patin '[PATI]'
      T     DBB [AR2, P#0.0];
      L     'PATI';
      T     DBD [AR2, P#1.0];
      L     ']';
      T     DBB [AR2, P#5.0];
      +AR2  P#6.0;

      L     "DB815_UTs_Datos".UT[#NumeroUT].GaliboPatin;
      T     #Valor;

// --- Convertir Valor a ASCII -  Patin
      TAR2;
      SRD   3;
      T     #NumBytes;  // Miro que offset tiene la String

      CALL  "FC893_Obtener_StringDelAtributo"
      ( DB_String := #NumDBEventos,
        OffsetIni := #NumBytes,
        Valor     := #Valor,
        OffsetFin := #Offset
      );  // Llamo a ObtenerStrinAtributo

      L     #Offset;
      SLD   3;
      LAR2;  // Recupero que offset tiene la String

// --- Ya esta convertido el Valor a ASCI - Fin Patin
CodigoPatin_DATO_EventoUT:NOP   0;



////////////////////////////////////////////////////////////////////////////////
// --- Atributo de ETIQUETA (Si es necesario) --- Router
      SET;  // Tiene Etiqueta ?
      AN    "DB850_DefinicionMesas".Mesa[#NumMesa].AtributosGalibo_DeEvento.EtiquetaRouter;
      JC    FinEtiquetaRouter_DATO_EventoUT;

      OPN   DB [#DBEventos];
      L     '[';  // Evento - Atributo Etiqueta '[SSCC]'
      T     DBB [AR2, P#0.0];
      L     'SSCC';
      T     DBD [AR2, P#1.0];
      L     ']';
      T     DBB [AR2, P#5.0];
      +AR2  P#6.0;

      L     0;  // Puntero a la Etiqueta
      T     #IndiceEtiqueta;

      L     "DB814_UTs_Etiqueta".UT[#NumeroUT].EtiquetaRouter;
      T     #Valor;  // Recoge el caracter de la Etiqueta

// --- Convertir Valor a ASCII -  Etiqueta Router
      TAR2;
      SRD   3;
      T     #NumBytes;  // Miro que offset tiene la String

      CALL  "FC893_Obtener_StringDelAtributo"
      ( DB_String := #NumDBEventos,
        OffsetIni := #NumBytes,
        Valor     := #Valor,
        OffsetFin := #Offset
      );  // Llamo a ObtenerStrinAtributo

      L     #Offset;
      SLD   3;
      LAR2;  // Recupero que offset tiene la String

// --- Ya esta convertido el Valor a ASCI - Fin Etiqueta Router
FinEtiquetaRouter_DATO_EventoUT:NOP   0;







////////////////////////////////////////////////////////////////////////////////
// --- Atributo de ETIQUETA (Si es necesario) --- STRING
      SET;  // Tiene Etiqueta ?
      AN    "DB850_DefinicionMesas".Mesa[#NumMesa].AtributosGalibo_DeEvento.EtiquetaString;
      JC    FinEtiquetaString_DATO_EventoUT;

      OPN   DB [#DBEventos];
      L     '[';  // Evento - Atributo Etiqueta '[SSCC]'
      T     DBB [AR2, P#0.0];
      L     'SSCC';
      T     DBD [AR2, P#1.0];
      L     ']';
      T     DBB [AR2, P#5.0];
      +AR2  P#6.0;

      L     2;  // Puntero a la Etiqueta
      T     #IndiceEtiqueta;

BucleEtiquetaString_DATO_EventoUT:NOP   0;
      L     "DB814_UTs_Etiqueta".UT[#NumeroUT].Etiqueta[#IndiceEtiqueta];
      T     #Valor;  // Recoge el caracter de la Etiqueta

      L     #Valor;
      L     0;
      ==I;
      JC    FinEtiquetaString_DATO_EventoUT;  // Es Final de Etiqueta?

      OPN   DB [#DBEventos];
      L     #Valor;
      T     DBB [AR2, P#0.0];

      L     #IndiceEtiqueta;  // Siguiente Caracter
      L     1;
      +I;
      T     #IndiceEtiqueta;
      +AR2  P#1.0;
      JU    BucleEtiquetaString_DATO_EventoUT;

FinEtiquetaString_DATO_EventoUT:NOP   0;





////////////////////////////////////////////////////////////////////////////////
// --- Final del Formato del Evento ---

      OPN   DB [#DBEventos];  // DB de Eventos Generados (A Emitir)
      L     '}';  // Fin de Evento '}'
      T     DBB [AR2, P#0.0];
      +AR2  P#1.0;


////////////////////////////////////////////////////////////////////////////////
////////////////////////////////////////////////////////////////////////////////
////////////////////////////////////////////////////////////////////////////////
////////////////////////////////////////////////////////////////////////////////
// Dar por formateado el Evento

      L     0;  // 0 - Dar por Tratado
      T     "DB812_UTs_Control".UT[#NumeroUT].EstadoEventoAGenerar;

////////////////////////////////////////////////////////////////////////////////
/// Hay que Pedir Datos
      SET;
      AN    "DB812_UTs_Control".UT[#NumeroUT].AtributosDeLaUT.PeticionDeDatos;
      JC    NoPedirDatos_DATO_EventosUT;

      L     141;
      T     "DB812_UTs_Control".UT[#NumeroUT].EstadoEventoAGenerar;

NoPedirDatos_DATO_EventosUT:NOP   0;


////////////////////////////////////////////////////////////////////////////////
      JU    FinBucles_EventosUT;


// Fin del formateo del Evento DATO
////////////////////////////////////////////////////////////////////////////////
////////////////////////////////////////////////////////////////////////////////
////////////////////////////////////////////////////////////////////////////////
////////////////////////////////////////////////////////////////////////////////



NETWORK
TITLE = ---- Evento de UT - Peticion de Datos de la UT - DAT?
GenerarEvento_DAT_EventosUT:NOP   0;

////////////////////////////////////////////////////////////////////////////////
////////////////////////////////////////////////////////////////////////////////
////////////////////////////////////////////////////////////////////////////////
// -- Formateo del Evento DAT? - Peticion de Datos para la UT
// -- Hay que poner que campo?       ¡¡¡ OJO !!!

      L     #P_Eventos;
      LAR2;  // Puntero al DB de Eventos Generados

      TAR2;  // Mirar si es el primer evento de la lista
      L     0;
      ==I;
      JC    InicioBuffer_DAT_EventosUT;  // Es el primero

      OPN   DB [#DBEventos];  // Hay que añadir si no es el primer evento
      L     ',';  // Separador entre eventos ','
      T     DBB [AR2, P#0.0];
      +AR2  P#1.0;

InicioBuffer_DAT_EventosUT:NOP   0;
      OPN   DB [#DBEventos];  // DB de Eventos Generados (A Emitir)
      L     '{';  // Inicio de Evento '{'
      T     DBB [AR2, P#0.0];
      +AR2  P#1.0;

      L     'DAT?';  // Evento 'DAT?'
      T     DBD [AR2, P#0.0];
      +AR2  P#4.0;


////////////////////////////////////////////////////////////////////////////////
      L     '[';  // Evento - Atributo Mckey '[MCKY]'
      T     DBB [AR2, P#0.0];
      L     'MCKY';
      T     DBD [AR2, P#1.0];
      L     ']';
      T     DBB [AR2, P#5.0];
      +AR2  P#6.0;

      L     "DB812_UTs_Control".UT[#NumeroUT].Mckey;
      T     #Valor;

// --- Convertir Valor a ASCII - Mckey
      TAR2;
      SRD   3;
      T     #NumBytes;  // Miro que offset tiene la String

      CALL  "FC893_Obtener_StringDelAtributo"
      ( DB_String := #NumDBEventos,
        OffsetIni := #NumBytes,
        Valor     := #Valor,
        OffsetFin := #Offset
      );  // Llamo a ObtenerStrinAtributo

      L     #Offset;
      SLD   3;
      LAR2;  // Recupero que offset tiene la String

// --- Ya esta convertido el Valor a ASCI - Fin Mckey


////////////////////////////////////////////////////////////////////////////////
      OPN   DB [#DBEventos];
      L     '[';  // Evento - Atributo Mesa Actual '[MESA]'
      T     DBB [AR2, P#0.0];
      L     'MESA';
      T     DBD [AR2, P#1.0];
      L     ']';
      T     DBB [AR2, P#5.0];
      +AR2  P#6.0;

      L     "DB812_UTs_Control".UT[#NumeroUT].MesaActual;
      T     #Valor;

// --- Convertir Valor a ASCII -  Mesa Actual
      TAR2;
      SRD   3;
      T     #NumBytes;  // Miro que offset tiene la String

      CALL  "FC893_Obtener_StringDelAtributo"
      ( DB_String := #NumDBEventos,
        OffsetIni := #NumBytes,
        Valor     := #Valor,
        OffsetFin := #Offset
      );  // Llamo a ObtenerStrinAtributo

      L     #Offset;
      SLD   3;
      LAR2;  // Recupero que offset tiene la String

// --- Ya esta convertido el Valor a ASCI - Fin Mesa Actual


////////////////////////////////////////////////////////////////////////////////
// --- Final del Formato del Evento ---

      OPN   DB [#DBEventos];  // DB de Eventos Generados (A Emitir)
      L     '}';  // Fin de Evento '}'
      T     DBB [AR2, P#0.0];
      +AR2  P#1.0;


////////////////////////////////////////////////////////////////////////////////
////////////////////////////////////////////////////////////////////////////////
////////////////////////////////////////////////////////////////////////////////
////////////////////////////////////////////////////////////////////////////////
// Dar por formateado el Evento

      L     0;  // 0 - Dar por Tratado
      T     "DB812_UTs_Control".UT[#NumeroUT].EstadoEventoAGenerar;

      SET;
      R     "DB812_UTs_Control".UT[#NumeroUT].AtributosDeLaUT.PeticionDeDatos;

      JU    FinBucles_EventosUT;

// Fin del formateo del Evento PD
////////////////////////////////////////////////////////////////////////////////
////////////////////////////////////////////////////////////////////////////////
////////////////////////////////////////////////////////////////////////////////
////////////////////////////////////////////////////////////////////////////////



NETWORK
TITLE = ---- Evento de UT - Chequeo de la UT - CHEQ!
GenerarEvento_CHE_EventosUT:NOP   0;

////////////////////////////////////////////////////////////////////////////////
////////////////////////////////////////////////////////////////////////////////
////////////////////////////////////////////////////////////////////////////////
// -- Formateo del Evento CHE! - Datos UT En Reset
// -- Hay que poner que campo?       ¡¡¡ OJO !!!

      L     #P_Eventos;
      LAR2;  // Puntero al DB de Eventos Generados

      TAR2;  // Mirar si es el primer evento de la lista
      L     0;
      ==I;
      JC    InicioBuffer_CHE_EventosUT;  // Es el primero

      OPN   DB [#DBEventos];  // Hay que añadir si no es el primer evento
      L     ',';  // Separador entre eventos ','
      T     DBB [AR2, P#0.0];
      +AR2  P#1.0;

InicioBuffer_CHE_EventosUT:NOP   0;
      OPN   DB [#DBEventos];  // DB de Eventos Generados (A Emitir)
      L     '{';  // Inicio de Evento '{'
      T     DBB [AR2, P#0.0];
      +AR2  P#1.0;

      L     'CHE!';  // Evento 'DAT?'
      T     DBD [AR2, P#0.0];
      +AR2  P#4.0;


////////////////////////////////////////////////////////////////////////////////
      OPN   DB [#DBEventos];
      L     '[';  // Evento - Atributo TIPO '[TIPO]'
      T     DBB [AR2, P#0.0];
      L     'TIPO';
      T     DBD [AR2, P#1.0];
      L     ']';
      T     DBB [AR2, P#5.0];
      +AR2  P#6.0;

      L     'MCKY';
      T     DBD [AR2, P#0.0];
      +AR2  P#4.0;


////////////////////////////////////////////////////////////////////////////////
      OPN   DB [#DBEventos];
      L     '[';  // Evento - Atributo Mckey '[NUME]'
      T     DBB [AR2, P#0.0];
      L     'NUME';
      T     DBD [AR2, P#1.0];
      L     ']';
      T     DBB [AR2, P#5.0];
      +AR2  P#6.0;

      L     "DB812_UTs_Control".UT[#NumeroUT].Mckey;
      T     #Valor;

// --- Convertir Valor a ASCII - Mckey
      TAR2;
      SRD   3;
      T     #NumBytes;  // Miro que offset tiene la String

      CALL  "FC893_Obtener_StringDelAtributo"
      ( DB_String := #NumDBEventos,
        OffsetIni := #NumBytes,
        Valor     := #Valor,
        OffsetFin := #Offset
      );  // Llamo a ObtenerStrinAtributo

      L     #Offset;
      SLD   3;
      LAR2;  // Recupero que offset tiene la String

// --- Ya esta convertido el Valor a ASCI - Fin Mckey


////////////////////////////////////////////////////////////////////////////////
      OPN   DB [#DBEventos];
      L     '[';  // Evento - Atributo Mesa Actual '[MESA]'
      T     DBB [AR2, P#0.0];
      L     'MESA';
      T     DBD [AR2, P#1.0];
      L     ']';
      T     DBB [AR2, P#5.0];
      +AR2  P#6.0;

      L     "DB812_UTs_Control".UT[#NumeroUT].MesaActual;
      T     #Valor;

// --- Convertir Valor a ASCII -  Mesa Actual
      TAR2;
      SRD   3;
      T     #NumBytes;  // Miro que offset tiene la String

      CALL  "FC893_Obtener_StringDelAtributo"
      ( DB_String := #NumDBEventos,
        OffsetIni := #NumBytes,
        Valor     := #Valor,
        OffsetFin := #Offset
      );  // Llamo a ObtenerStrinAtributo

      L     #Offset;
      SLD   3;
      LAR2;  // Recupero que offset tiene la String

// --- Ya esta convertido el Valor a ASCI - Fin Mesa Actual


////////////////////////////////////////////////////////////////////////////////
      OPN   DB [#DBEventos];
      L     '[';  // Evento - Atributo Resultado '[RESU]'
      T     DBB [AR2, P#0.0];
      L     'RESU';
      T     DBD [AR2, P#1.0];
      L     ']';
      T     DBB [AR2, P#5.0];
      +AR2  P#6.0;

      L     'TRUE';
      T     DBD [AR2, P#0.0];
      +AR2  P#4.0;


////////////////////////////////////////////////////////////////////////////////
// --- Final del Formato del Evento ---

      OPN   DB [#DBEventos];  // DB de Eventos Generados (A Emitir)
      L     '}';  // Fin de Evento '}'
      T     DBB [AR2, P#0.0];
      +AR2  P#1.0;


////////////////////////////////////////////////////////////////////////////////
////////////////////////////////////////////////////////////////////////////////
////////////////////////////////////////////////////////////////////////////////
////////////////////////////////////////////////////////////////////////////////
// Dar por formateado el Evento

      L     0;  // 0 - Dar por Tratado
      T     "DB812_UTs_Control".UT[#NumeroUT].EstadoEventoAGenerar;

      JU    FinBucles_EventosUT;

// Fin del formateo del Evento PD
////////////////////////////////////////////////////////////////////////////////
////////////////////////////////////////////////////////////////////////////////
////////////////////////////////////////////////////////////////////////////////
////////////////////////////////////////////////////////////////////////////////



NETWORK
TITLE = ---- Evento de UT - Peticion de Datos de Embandejado - PEMB // Fecha 07 06 2017
GenerarEvento_PEMB_EventosUT:NOP   0;

////////////////////////////////////////////////////////////////////////////////
////////////////////////////////////////////////////////////////////////////////
///////////////////////////////////////////////////////////////////////////////
// -- Formateo del Evento PEMB (Peticion de Datos de Embandejado de la UT)

      L     #P_Eventos;
      LAR2;  // Puntero al DB de Eventos Generados

      TAR2;  // Mirar si es el primer evento de la lista
      L     0;
      ==I;
      JC    InicioBuffer_PEMB_EventosUT;  // Es el primero

      OPN   DB [#DBEventos];  // Hay que añadir si no es el primer evento
      L     ',';  // Separador entre eventos ','
      T     DBB [AR2, P#0.0];
      +AR2  P#1.0;

InicioBuffer_PEMB_EventosUT:NOP   0;
      OPN   DB [#DBEventos];  // DB de Eventos Generados (A Emitir)
      L     '{';  // Inicio de Evento '{'
      T     DBB [AR2, P#0.0];
      +AR2  P#1.0;

      L     'PEMB';  // Evento 'PEMB'
      T     DBD [AR2, P#0.0];
      +AR2  P#4.0;


////////////////////////////////////////////////////////////////////////////////
      L     '[';  // Evento - Atributo Mckey '[MCKY]'
      T     DBB [AR2, P#0.0];
      L     'MCKY';
      T     DBD [AR2, P#1.0];
      L     ']';  // Evento - Atributo Mckey '[MCKY]'
      T     DBB [AR2, P#5.0];
      +AR2  P#6.0;

      L     "DB812_UTs_Control".UT[#NumeroUT].Mckey;
      T     #Valor;

// --- Convertir Valor a ASCII - Mckey
      TAR2;
      SRD   3;
      T     #NumBytes;  // Miro que offset tiene la String

      CALL  "FC893_Obtener_StringDelAtributo"
      ( DB_String := #NumDBEventos,
        OffsetIni := #NumBytes,
        Valor     := #Valor,
        OffsetFin := #Offset
      );  // Llamo a ObtenerStrinAtributo

      L     #Offset;
      SLD   3;
      LAR2;  // Recupero que offset tiene la String

// --- Ya esta convertido el Valor a ASCI - Fin Mckey


///////////////////////////////////////////////////////////////////////////////
      OPN   DB [#DBEventos];
      L     '[';  // Evento - Atributo Mesa Actual '[MESA]'
      T     DBB [AR2, P#0.0];
      L     'MESA';
      T     DBD [AR2, P#1.0];
      L     ']';
      T     DBB [AR2, P#5.0];
      +AR2  P#6.0;

      L     "DB812_UTs_Control".UT[#NumeroUT].MesaActual;
      T     #Valor;

// --- Convertir Valor a ASCII -  Mesa Actual
      TAR2;
      SRD   3;
      T     #NumBytes;  // Miro que offset tiene la String

      CALL  "FC893_Obtener_StringDelAtributo"
      ( DB_String := #NumDBEventos,
        OffsetIni := #NumBytes,
        Valor     := #Valor,
        OffsetFin := #Offset
      );  // Llamo a ObtenerStrinAtributo

      L     #Offset;
      SLD   3;
      LAR2;  // Recupero que offset tiene la String

// --- Ya esta convertido el Valor a ASCI - Fin Mesa Actual


///////////////////////////////////////////////////////////////////////////////
// --- Final del Formateo del Evento ---

      OPN   DB [#DBEventos];  // DB de Eventos Generados (A Emitir)
      L     '}';  // Fin de Evento '}'
      T     DBB [AR2, P#0.0];
      +AR2  P#1.0;

///////////////////////////////////////////////////////////////////////////////
///////////////////////////////////////////////////////////////////////////////
///////////////////////////////////////////////////////////////////////////////
// Dar por formateado el Evento

      L     0;  // 0 - Dar por Tratado
      T     "DB812_UTs_Control".UT[#NumeroUT].EstadoEventoAGenerar;

      JU    FinBucles_EventosUT;

// Fin del Evento PEMB
///////////////////////////////////////////////////////////////////////////////
///////////////////////////////////////////////////////////////////////////////
///////////////////////////////////////////////////////////////////////////////



NETWORK
TITLE = Generar Eventos de las Mesas
// Recorrer toda las Mesas (Dispositivos)
// Si el Campo EstadoEmision >= 100 se ha generado un evento
EventosMesa:NOP   0;

////////////////////////////////////////////////////////////////////////////////
////////////////////////////////////////////////////////////////////////////////
////////////////////////////////////////////////////////////////////////////////
// - Recorrer todas las Mesas

      L     #InicioBucleMesas;
      T     #NumMesa;

InicioBucle_EventosMesa:NOP   0;
////////////////////////////////////////////////////////////////////////////////
/// Mirar Si pertenece al JDT

      SET;
      X     "DB850_DefinicionMesas".Mesa[#NumMesa].ConfigMesa.MesaDeJDT02;  // JDT01 ?
      XN    #JDT02_Activo;
      =     #MesaDeJDT02;

      SET;
      AN    #MesaDeJDT02;
      JC    ContinuarBucle_EventosMesa;

////////////////////////////////////////////////////////////////////////////////
/// Mirar si esta definido como mesa de Tracking y TL

      SET;
      AN    "DB850_DefinicionMesas".Mesa[#NumMesa].ConfigMesa.MesaPaso;
      AN    "DB850_DefinicionMesas".Mesa[#NumMesa].ConfigMesa.MesaCruce;
      AN    "DB850_DefinicionMesas".Mesa[#NumMesa].ConfigMesa.MesaMultiplesDestinos;
      AN    "DB850_DefinicionMesas".Mesa[#NumMesa].ConfigMesa.MesaTL;
      JC    ContinuarBucle_EventosMesa;


////////////////////////////////////////////////////////////////////////////////

      L     "DB831_Mesas".Mesas[#NumMesa].EstadoEmisionEvento;
      T     #EventoDispositivo;  // Posicion 2

      L     #EventoDispositivo;
      L     100;  // Mirar si hay Evento a Generar
      >=I;  // >= 100 Hay Evento Generado
      JC    Generar_EventosMesa;


////////////////////////////////////////////////////////////////////////////////
// - Continuar con la Suquiente Mesa
ContinuarBucle_EventosMesa:NOP   0;
      L     #NumMesa;  // Si no hay más dispositivos Mesas
      L     #FinalBucleMesas;
      >=I;
      JC    FinalFuncion;  // Ya no hay más dispositivos Mesas, Finalizar

      L     #NumMesa;  // +1, Para la Siguiente Mesa
      L     1;
      +I;
      T     #NumMesa;
      JU    InicioBucle_EventosMesa;

////////////////////////////////////////////////////////////////////////////////
// Comprobacion del tamaño del DB de Eventos Generados
FinBucle_EventosMesa:NOP   0;
      TAR2;
      T     #P_Eventos;
      SRD   3;
      T     #NumBytes;

      L     #NumBytes;  // Miramos si hay sitio
      L     #MaxBytes;
      >I;
      JC    FinalFuncion;  // No se pueden generar más eventos
      JU    ContinuarBucle_EventosMesa;  // Ya se ha generado los eventos de dispositivos mesas



NETWORK
TITLE = Formatear Eventos de las Mesas - Distribucion
// - Distribucion para Eventos de las Mesas
// - Formateo de Eventos
//   - Evento STAT (Cambio de Estado del Dispositivo)
//   - Evento FIN! (Proceso del Dispositivo Finalizado)
//   - Evento DIS? (Pedir datos del Dispositivo)
Generar_EventosMesa:NOP   0;

////////////////////////////////////////////////////////////////////////////////
////////////////////////////////////////////////////////////////////////////////
// -- Formateo del Evento STAT (Estado del Dispositivo)
// -- Formateo del Evento FIN! (Fin del Proceso --> Reset y Paro Blando)
// -- Formateo del Evento DIS? (Peticion de Estado del Dispositivo)
////////////////////////////////////////////////////////////////////////////////
////////////////////////////////////////////////////////////////////////////////
// - Distrubucion de Generarcion de Eventos

      L     #EventoDispositivo;
      L     160;  // Formateo del Evento
      ==I;  // Refresco de datos de la Mesa
      JC    GenerarEvento_STAT_EventosMesa;

      L     #EventoDispositivo;
      L     161;  // Formateo del evento
      ==I;  // Peticion de Datos del Dispositivo
      JC    GenerarEvento_DIS_EventosMesa;

      L     #EventoDispositivo;
      L     151;  // Formateo del Evento
      ==I;  // Fin de Reset OK
      JC    GenerarEvento_FIN_EventosMesa;

      L     #EventoDispositivo;
      L     152;  // Formateo del Evento
      ==I;  // Fin de Reset NOK
      JC    GenerarEvento_FIN_EventosMesa;

      L     #EventoDispositivo;
      L     153;  // Formateo del Evento
      ==I;  // Fin Paro Blando OK
      JC    GenerarEvento_FIN_EventosMesa;

      L     #EventoDispositivo;
      L     154;  // Formateo del Evento
      ==I;  // Fin Paro Blando NOK
      JC    GenerarEvento_FIN_EventosMesa;


////////////////////////////////////////////////////////////////////////////////
////////////////////////////////////////////////////////////////////////////////
// --- Dar por formateado el Evento
// --- No existe el Evento

      L     0;  // Lo doy por tratado
      T     "DB831_Mesas".Mesas[#NumMesa].EstadoEmisionEvento;

      JU    FinBucle_EventosMesa;  // No existe ese tipo de Evento



NETWORK
TITLE = --- Evento de Dispositivo Mesa - Estado de Dispositivo - STAT
////////////////////////////////////////////////////////////////////////////////
////////////////////////////////////////////////////////////////////////////////
////////////////////////////////////////////////////////////////////////////////
// -- Formateo del Evento STAT (Estado del Dispositivo)
GenerarEvento_STAT_EventosMesa:NOP   0;

      L     #P_Eventos;
      LAR2;  // Puntero al DB de Eventos Generados

      TAR2;  // Mirar si es el primer evento de la lista
      L     0;
      ==I;
      JC    InicioBuffer_STAT_EventosMesa;  // Es el primero

      OPN   DB [#DBEventos];
      L     ',';  // Separador entre eventos ','
      T     DBB [AR2, P#0.0];
      +AR2  P#1.0;

InicioBuffer_STAT_EventosMesa:NOP   0;
      OPN   DB [#DBEventos];  // DB de Eventos Generados (A Emitir)
      L     '{';  // Inicio de Evento '{'
      T     DBB [AR2, P#0.0];
      +AR2  P#1.0;

      L     'STAT';  // Evento 'STAT'
      T     DBD [AR2, P#0.0];
      +AR2  P#4.0;


////////////////////////////////////////////////////////////////////////////////
      OPN   DB [#DBEventos];
      L     '[';  // Evento - Atributo Tipo '[TIPO]'
      T     DBB [AR2, P#0.0];
      L     'TIPO';
      T     DBD [AR2, P#1.0];
      L     ']';
      T     DBB [AR2, P#5.0];
      +AR2  P#6.0;

      L     60;  // Dispo Mesa
      T     #Convertir;
      CALL  "FC895_Obtener_EtiquetaDeValor"
      ( ValorEvento    := #Convertir,
        EtiquetaEvento := #Conversion
      );

      OPN   DB [#DBEventos];
      L     #Conversion;
      T     DBD [AR2, P#0.0];
      +AR2  P#4.0;


////////////////////////////////////////////////////////////////////////////////
      L     '[';  // Evento - Atributo Numero de Dispositivo '[NUME]'
      T     DBB [AR2, P#0.0];
      L     'NUME';
      T     DBD [AR2, P#1.0];
      L     ']';
      T     DBB [AR2, P#5.0];
      +AR2  P#6.0;

      L     "CTE_OffsetMesa";
      L     #NumMesa;  // Numero de Mesa
      +I;
      T     #Valor;

// --- Convertir Valor a ASCII - Numero de Mesa
      TAR2;
      SRD   3;
      T     #NumBytes;  // Miro que offset tiene la String

      CALL  "FC893_Obtener_StringDelAtributo"
      ( DB_String := #NumDBEventos,
        OffsetIni := #NumBytes,
        Valor     := #Valor,
        OffsetFin := #Offset
      );  // Llamo a ObtenerStrinAtributo

      L     #Offset;
      SLD   3;
      LAR2;  // Recupero que offset tiene la String

// --- Ya esta convertido el Valor a ASCII


////////////////////////////////////////////////////////////////////////////////
      OPN   DB [#DBEventos];
      L     '[';  // Evento - Atributo Numero de Dispositivo '[NUES]'
      T     DBB [AR2, P#0.0];
      L     'NUES';
      T     DBD [AR2, P#1.0];
      L     ']';
      T     DBB [AR2, P#5.0];
      +AR2  P#6.0;

      L     "DB831_Mesas".Mesas[#NumMesa].StatusActual;
      L     W#16#F;  // Solo la parte Estado
      AW;
      T     #Convertir;

      CALL  "FC895_Obtener_EtiquetaDeValor"
      ( ValorEvento    := #Convertir,
        EtiquetaEvento := #Conversion
      );

      OPN   DB [#DBEventos];
      L     #Conversion;
      T     DBD [AR2, P#0.0];
      +AR2  P#4.0;


